// TIA Portal V15.1 export
// export: Created 2024-06-21T08:41:20.6972322Z, ExportSetting WithDefaults, DisplayName Totally Integrated Automation Portal, DisplayVersion V15.1 Update 5, DisplayName TIA Portal Openness, DisplayVersion V15.1 Update 5, DisplayName SINAMICS Startdrive Advanced, DisplayVersion V15.1, DisplayName G130, G150, S120, S150, SINAMICS MV, S210, DisplayVersion V15.1, DisplayName G110M, G120, G120C, G120D, G120P, DisplayVersion V15.1, DisplayName STEP 7 Professional, DisplayVersion V15.1 Update 5, DisplayName STEP 7 Safety, DisplayVersion V15.1, DisplayName WinCC Professional, DisplayVersion V15.1 Update 5, DisplayName SIMATIC Visualization Architect, DisplayVersion V15.1
FUNCTION_BLOCK "LCycleMonitoring"   // FB6056, FBD
TITLE = LCycleMonitoring - 2017/08/31
{ S7_Optimized_Access := 'FALSE' }
AUTHOR : hbracke
FAMILY : DataHand
VERSION : 0.1
// Used to monitor the cycle of a subzone and report the results to IT. On top it also creates an overtime alarm.
// stored: AutoNumber false, IsIECCheckEnabled false, SetENOAutomatically False, UDAEnableTagReadback false
   VAR_INPUT
      I_DateTimeFromPlc { ExternalAccessible := 'False'; ExternalVisible := 'False'; ExternalWritable := 'False'} : Date_And_Time;   // Actual Date and time from PLC
      I_PlcStatus { ExternalAccessible := 'False'; ExternalVisible := 'False'; ExternalWritable := 'False'} : DWord;   // Actual global PLC status
      I_ZmStatus { ExternalAccessible := 'False'; ExternalVisible := 'False'; ExternalWritable := 'False'} : "ZMStatus";   // Actual ModeZone status
      I_SubZoneStatus { ExternalAccessible := 'False'; ExternalVisible := 'False'; ExternalWritable := 'False'} : "SubzoneStatus";   // Actual status of one Subzone within the ModeZone
      I_OperatorStatus1 { ExternalAccessible := 'False'; ExternalVisible := 'False'; ExternalWritable := 'False'} : "OperatorStatus";   // Actual status of an operator
      I_OperatorStatus2 { ExternalAccessible := 'False'; ExternalVisible := 'False'; ExternalWritable := 'False'} : "OperatorStatus";   // Actual status of an operator
      I_OperatorStatus3 { ExternalAccessible := 'False'; ExternalVisible := 'False'; ExternalWritable := 'False'} : "OperatorStatus";   // Actual status of an operator
      I_OperatorStatus4 { ExternalAccessible := 'False'; ExternalVisible := 'False'; ExternalWritable := 'False'} : "OperatorStatus";   // Actual status of an operator
      I_OperatorStatus5 { ExternalAccessible := 'False'; ExternalVisible := 'False'; ExternalWritable := 'False'} : "OperatorStatus";   // Actual status of an operator
      I_OperatorStatus6 { ExternalAccessible := 'False'; ExternalVisible := 'False'; ExternalWritable := 'False'} : "OperatorStatus";   // Actual status of an operator
      I_PcsBodyId { ExternalAccessible := 'False'; ExternalVisible := 'False'; ExternalWritable := 'False'} : DWord;   // Body identification of in the SubZone; can be BodyNumber, Tagnumber, MixNumber or sequence number
      I_PcsBodyType { ExternalAccessible := 'False'; ExternalVisible := 'False'; ExternalWritable := 'False'} : DWord;   // Body type identification in Subzone
      I_RobotProgramNumber { ExternalAccessible := 'False'; ExternalVisible := 'False'; ExternalWritable := 'False'} : DWord;   // Program number of the robot
      I_CarrierId { ExternalAccessible := 'False'; ExternalVisible := 'False'; ExternalWritable := 'False'} : DWord;   // Identification of the carrier
      I_SubCarrierId { ExternalAccessible := 'False'; ExternalVisible := 'False'; ExternalWritable := 'False'} : DWord;   // Identification of a subcarrier
      I_AutoZoneReferenceCycle { ExternalAccessible := 'False'; ExternalVisible := 'False'; ExternalWritable := 'False'} : DWord;   // Reference cycle time for this zone for this product type
      I_Operator1RefCycle { ExternalAccessible := 'False'; ExternalVisible := 'False'; ExternalWritable := 'False'} : DWord;   // Reference cycle time for this zone for this product type
      I_Operator2RefCycle { ExternalAccessible := 'False'; ExternalVisible := 'False'; ExternalWritable := 'False'} : DWord;   // Reference cycle time for this zone for this product type
      I_Operator3RefCycle { ExternalAccessible := 'False'; ExternalVisible := 'False'; ExternalWritable := 'False'} : DWord;   // Reference cycle time for this zone for this product type
      I_Operator4RefCycle { ExternalAccessible := 'False'; ExternalVisible := 'False'; ExternalWritable := 'False'} : DWord;   // Reference cycle time for this zone for this product type
      I_Operator5RefCycle { ExternalAccessible := 'False'; ExternalVisible := 'False'; ExternalWritable := 'False'} : DWord;   // Reference cycle time for this zone for this product type
      I_Operator6RefCycle { ExternalAccessible := 'False'; ExternalVisible := 'False'; ExternalWritable := 'False'} : DWord;   // Reference cycle time for this zone for this product type
      C_StationNumber { ExternalAccessible := 'False'; ExternalVisible := 'False'; ExternalWritable := 'False'} : DWord;   // Station number (6 digits) where this subzone belongs to. Syntax is LLLSSS where LLL is the line number and SSS is the station number.
      C_ModeZoneNumber { ExternalAccessible := 'False'; ExternalVisible := 'False'; ExternalWritable := 'False'} : DWord;   // Number of the modezone. LLLSSSZMxx where xx is the number of the modezone.
      C_SubZoneNumber { ExternalAccessible := 'False'; ExternalVisible := 'False'; ExternalWritable := 'False'} : DWord;   // Is a number identifying the subzone within the Modezone. Syntax is mmx where mm is the number of the modezone and x is a sequencial number of the subzone.
      C_SubSystem { ExternalAccessible := 'False'; ExternalVisible := 'False'; ExternalWritable := 'False'} : Int;   // Number to identify the subsystem / Identify Subsystem / Identification of the Subsystem
      C_VDCommRecvDB { ExternalAccessible := 'False'; ExternalVisible := 'False'; ExternalWritable := 'False'} : DB_ANY;   // VD communication system receive DB; Not to be used by Application
      C_VDCommSendDB { ExternalAccessible := 'False'; ExternalVisible := 'False'; ExternalWritable := 'False'} : DB_ANY;   // VD communication system send DB; Not to be used by Application
      C_LocalRecvDB { ExternalAccessible := 'False'; ExternalVisible := 'False'; ExternalWritable := 'False'} : DB_ANY;   // Local DB For Recv Data Used By The Application
      C_LocalSendDB { ExternalAccessible := 'False'; ExternalVisible := 'False'; ExternalWritable := 'False'} : DB_ANY;   // Local DB For Send Data Used By The Application
   END_VAR
   VAR_OUTPUT
      O_WaitingInput { ExternalAccessible := 'False'; ExternalVisible := 'False'; ExternalWritable := 'False'} : Bool;   // Summary of waiting input status; any waiting input is active
      O_WaitingOutput { ExternalAccessible := 'False'; ExternalVisible := 'False'; ExternalWritable := 'False'} : Bool;   // Summary of waiting output status is active
      O_AutoZoneOverCycle { ExternalAccessible := 'False'; ExternalVisible := 'False'; ExternalWritable := 'False'} : Bool;   // Automatic unit has exceeded reference time
      O_Operator1OverCycle { ExternalAccessible := 'False'; ExternalVisible := 'False'; ExternalWritable := 'False'} : Bool;   // Operator has exceeded reference time
      O_Operator1OverCycleWarning { ExternalAccessible := 'False'; ExternalVisible := 'False'; ExternalWritable := 'False'} : Bool;   // Operator has exceeded 90% reference time
      O_Operator2OverCycle { ExternalAccessible := 'False'; ExternalVisible := 'False'; ExternalWritable := 'False'} : Bool;   // Operator has exceeded reference time
      O_Operator2OverCycleWarning { ExternalAccessible := 'False'; ExternalVisible := 'False'; ExternalWritable := 'False'} : Bool;   // Operator has exceeded 90% reference time
      O_Operator3OverCycle { ExternalAccessible := 'False'; ExternalVisible := 'False'; ExternalWritable := 'False'} : Bool;   // Operator has exceeded reference time
      O_Operator3OverCycleWarning { ExternalAccessible := 'False'; ExternalVisible := 'False'; ExternalWritable := 'False'} : Bool;   // Operator has exceeded 90% reference time
      O_Operator4OverCycle { ExternalAccessible := 'False'; ExternalVisible := 'False'; ExternalWritable := 'False'} : Bool;   // Operator has exceeded reference time
      O_Operator4OverCycleWarning { ExternalAccessible := 'False'; ExternalVisible := 'False'; ExternalWritable := 'False'} : Bool;   // Operator has exceeded 90% reference time
      O_Operator5OverCycle { ExternalAccessible := 'False'; ExternalVisible := 'False'; ExternalWritable := 'False'} : Bool;   // Operator has exceeded reference time
      O_Operator5OverCycleWarning { ExternalAccessible := 'False'; ExternalVisible := 'False'; ExternalWritable := 'False'} : Bool;   // Operator has exceeded 90% reference time
      O_Operator6OverCycle { ExternalAccessible := 'False'; ExternalVisible := 'False'; ExternalWritable := 'False'} : Bool;   // Operator has exceeded reference time
      O_Operator6OverCycleWarning { ExternalAccessible := 'False'; ExternalVisible := 'False'; ExternalWritable := 'False'} : Bool;   // Operator has exceeded 90% reference time
      O_WarningAlarm { ExternalAccessible := 'False'; ExternalVisible := 'False'; ExternalWritable := 'False'} : Bool;   // Summary of internal warning alarms
   END_VAR
   VAR_IN_OUT
      IO_VD : "VDComm";   // Signal handshake LVdComMaster
      IO_Modes : "Modes";   // Modes record to infeed the modes status of this subzone
      IO_Robot1 : "Robot";   // Robot record to exchange all robot statusses
      IO_Robot2 : "Robot";   // Robot record to exchange all robot statusses
      IO_Robot3 : "Robot";   // Robot record to exchange all robot statusses
      IO_Robot4 : "Robot";   // Robot record to exchange all robot statusses
      IO_Robot5 : "Robot";   // Robot record to exchange all robot statusses
      IO_Robot6 : "Robot";   // Robot record to exchange all robot statusses
      IO_Robot7 : "Robot";   // Robot record to exchange all robot statusses
      IO_Robot8 : "Robot";   // Robot record to exchange all robot statusses
      IO_Robot9 : "Robot";   // Robot record to exchange all robot statusses
      IO_Robot10 : "Robot";   // Robot record to exchange all robot statusses
      IO_Robot11 : "Robot";   // Robot record to exchange all robot statusses
      IO_Robot12 : "Robot";   // Robot record to exchange all robot statusses
      IO_Robot13 : "Robot";   // Robot record to exchange all robot statusses
      IO_Robot14 : "Robot";   // Robot record to exchange all robot statusses
      H_HMI : "H_HMI";   // HMI interface
      H_CycleMonitor : "H_CycleMonitoring";   // HMI interface
   END_VAR
   VAR DB_SPECIFIC
      DateTime { ExternalAccessible := 'False'; ExternalVisible := 'False'; ExternalWritable := 'False'} : Date_And_Time;   // Date and Time from the PLC. Each scan updated.
      SendToVD { ExternalAccessible := 'False'; ExternalVisible := 'False'; ExternalWritable := 'False'} : Bool;   // Trigger to send data to VD when Cycle is finished
      SendDoneVD { ExternalAccessible := 'False'; ExternalVisible := 'False'; ExternalWritable := 'False'} : Bool;   // Request Is Finished / Send operation is finished
      ResetVDComm { ExternalAccessible := 'False'; ExternalVisible := 'False'; ExternalWritable := 'False'} : Bool;   // Reset VD communication upon timeout
      InitState { ExternalAccessible := 'False'; ExternalVisible := 'False'; ExternalWritable := 'False'} : Bool;   // Flag indicating the initial run of the module
      StartOfCyclePulse { ExternalAccessible := 'False'; ExternalVisible := 'False'; ExternalWritable := 'False'} : Bool;   // Pulse at the start of a cycle
      EndOfCyclePulse { ExternalAccessible := 'False'; ExternalVisible := 'False'; ExternalWritable := 'False'} : Bool;   // Pulse at end of the cycle
      EndOfCycleReached { ExternalAccessible := 'False'; ExternalVisible := 'False'; ExternalWritable := 'False'} : Bool;   // Bit set to indicate the end of a cycle
      EndOfRecordReached { ExternalAccessible := 'False'; ExternalVisible := 'False'; ExternalWritable := 'False'} : Bool;   // Bit set when end of record was reached. A new record shall be setup
      AnyRobotActive { ExternalAccessible := 'False'; ExternalVisible := 'False'; ExternalWritable := 'False'} : Bool;   // Summary of all robots active
      AnyOperatorActive { ExternalAccessible := 'False'; ExternalVisible := 'False'; ExternalWritable := 'False'} : Bool;   // Summary of all operators active
      AnyOperatorOverCycle { ExternalAccessible := 'False'; ExternalVisible := 'False'; ExternalWritable := 'False'} : Bool;   // Summary of all operators
      StopActive { ExternalAccessible := 'False'; ExternalVisible := 'False'; ExternalWritable := 'False'} : Bool;   // Summery of all stopping conditions
      AutoZoneOverCycle { ExternalAccessible := 'False'; ExternalVisible := 'False'; ExternalWritable := 'False'} : Bool;   // Automatic zone is in over cycle
      WaitingInput { ExternalAccessible := 'False'; ExternalVisible := 'False'; ExternalWritable := 'False'} : Bool;   // Summary of all waiting input conditions
      WaitingOutput { ExternalAccessible := 'False'; ExternalVisible := 'False'; ExternalWritable := 'False'} : Bool;   // Summary of all waiting output conditions
      Operator1OverCycle { ExternalAccessible := 'False'; ExternalVisible := 'False'; ExternalWritable := 'False'} : Bool;   // Operator action exceeds reference tme
      Operator2OverCycle { ExternalAccessible := 'False'; ExternalVisible := 'False'; ExternalWritable := 'False'} : Bool;   // Operator action exceeds reference tme
      Operator3OverCycle { ExternalAccessible := 'False'; ExternalVisible := 'False'; ExternalWritable := 'False'} : Bool;   // Operator action exceeds reference tme
      Operator4OverCycle { ExternalAccessible := 'False'; ExternalVisible := 'False'; ExternalWritable := 'False'} : Bool;   // Operator action exceeds reference tme
      Operator5OverCycle { ExternalAccessible := 'False'; ExternalVisible := 'False'; ExternalWritable := 'False'} : Bool;   // Operator action exceeds reference tme
      Operator6OverCycle { ExternalAccessible := 'False'; ExternalVisible := 'False'; ExternalWritable := 'False'} : Bool;   // Operator action exceeds reference tme
      Operator1OverCycleWarning { ExternalAccessible := 'False'; ExternalVisible := 'False'; ExternalWritable := 'False'} : Bool;   // Operator action exceeds 90% of reference tme
      Operator2OverCycleWarning { ExternalAccessible := 'False'; ExternalVisible := 'False'; ExternalWritable := 'False'} : Bool;   // Operator action exceeds 90% of reference tme
      Operator3OverCycleWarning { ExternalAccessible := 'False'; ExternalVisible := 'False'; ExternalWritable := 'False'} : Bool;   // Operator action exceeds 90% of reference tme
      Operator4OverCycleWarning { ExternalAccessible := 'False'; ExternalVisible := 'False'; ExternalWritable := 'False'} : Bool;   // Operator action exceeds 90% of reference tme
      Operator5OverCycleWarning { ExternalAccessible := 'False'; ExternalVisible := 'False'; ExternalWritable := 'False'} : Bool;   // Operator action exceeds 90% of reference tme
      Operator6OverCycleWarning { ExternalAccessible := 'False'; ExternalVisible := 'False'; ExternalWritable := 'False'} : Bool;   // Operator action exceeds 90% of reference tme
      MaxRecordCountAlm { ExternalAccessible := 'False'; ExternalVisible := 'False'; ExternalWritable := 'False'} : Bool;   // Maximum amount of records within one cycle reported
      WarningAlarm { ExternalAccessible := 'False'; ExternalVisible := 'False'; ExternalWritable := 'False'} : Bool;   // Summary of warning alarms
      AlarmA { ExternalAccessible := 'False'; ExternalVisible := 'False'; ExternalWritable := 'False'} : Bool;   // Alarm A created by this function
      AlarmB { ExternalAccessible := 'False'; ExternalVisible := 'False'; ExternalWritable := 'False'} : Bool;   // Alarm B created by this function
      AlarmC { ExternalAccessible := 'False'; ExternalVisible := 'False'; ExternalWritable := 'False'} : Bool;   // Alarm C created by this function
      AlarmD { ExternalAccessible := 'False'; ExternalVisible := 'False'; ExternalWritable := 'False'} : Bool;   // Alarm D created by this function
      MaxIndex { ExternalAccessible := 'False'; ExternalVisible := 'False'; ExternalWritable := 'False'} : Int;   // Maximum value for Index
      Index { ExternalAccessible := 'False'; ExternalVisible := 'False'; ExternalWritable := 'False'} : Int;   // index to point to data values in event array
      MaxEofRecCounter { ExternalAccessible := 'False'; ExternalVisible := 'False'; ExternalWritable := 'False'} : Int;   // Maximum value that the record is allowed to loop without new start of cycle
      EofRecordCounter { ExternalAccessible := 'False'; ExternalVisible := 'False'; ExternalWritable := 'False'} : Int;   // Counting number of end of record events within 1 cycle
      SendLength { ExternalAccessible := 'False'; ExternalVisible := 'False'; ExternalWritable := 'False'} : Word;   // Pointer / Lenght of the data packet to be send
      VirtualBodyId { ExternalAccessible := 'False'; ExternalVisible := 'False'; ExternalWritable := 'False'} : DWord;   // Virtual created BodyId in case I_PcsBodyId is 0
      TotalProcessCycleTime { ExternalAccessible := 'False'; ExternalVisible := 'False'; ExternalWritable := 'False'} : Time;   // Accumulating timer (ms) to set the total cycle time
      TotalProcessWorkTime { ExternalAccessible := 'False'; ExternalVisible := 'False'; ExternalWritable := 'False'} : Time;   // Accumulating timer (ms) to set the total processwork time
      TotalOperator1Time { ExternalAccessible := 'False'; ExternalVisible := 'False'; ExternalWritable := 'False'} : Time;   // Accumulating timer (ms) of operator 1
      TotalOperator2Time { ExternalAccessible := 'False'; ExternalVisible := 'False'; ExternalWritable := 'False'} : Time;   // Accumulating timer (ms) of operator 2
      TotalOperator3Time { ExternalAccessible := 'False'; ExternalVisible := 'False'; ExternalWritable := 'False'} : Time;   // Accumulating timer (ms) of operator 3
      TotalOperator4Time { ExternalAccessible := 'False'; ExternalVisible := 'False'; ExternalWritable := 'False'} : Time;   // Accumulating timer (ms) of operator 4
      TotalOperator5Time { ExternalAccessible := 'False'; ExternalVisible := 'False'; ExternalWritable := 'False'} : Time;   // Accumulating timer (ms) of operator 5
      TotalOperator6Time { ExternalAccessible := 'False'; ExternalVisible := 'False'; ExternalWritable := 'False'} : Time;   // Accumulating timer (ms) of operator 6
      TotalWaitingInputTime { ExternalAccessible := 'False'; ExternalVisible := 'False'; ExternalWritable := 'False'} : Time;   // Accumulating timer (ms) to set the total waiting input time
      TotalInfeedTime { ExternalAccessible := 'False'; ExternalVisible := 'False'; ExternalWritable := 'False'} : Time;   // Accumulating timer (ms) to set the total Infeed time
      TotalWaitingOutputTime { ExternalAccessible := 'False'; ExternalVisible := 'False'; ExternalWritable := 'False'} : Time;   // Accumulating timer (ms) to set the total waiting output time
      TotalOutfeedTime { ExternalAccessible := 'False'; ExternalVisible := 'False'; ExternalWritable := 'False'} : Time;   // Accumulating timer (ms) to set the total Outfeed time
      TotalWaitingProcessWorkTime { ExternalAccessible := 'False'; ExternalVisible := 'False'; ExternalWritable := 'False'} : Time;   // Accumulating timer (ms) to set the total waiting process work time
      TotalWaitingRecoveryTime { ExternalAccessible := 'False'; ExternalVisible := 'False'; ExternalWritable := 'False'} : Time;   // Accumulating timer (ms) to set the total recovery time
      Memory { ExternalAccessible := 'False'; ExternalVisible := 'False'; ExternalWritable := 'False'} : Array[1..256] of Bool;   // Memory bits used to create edges
      CycleMonitorBuffer { ExternalAccessible := 'False'; ExternalVisible := 'False'; ExternalWritable := 'False'; S7_SetPoint := 'True'} : "H_CycleMonitoring";   // Array of display lines used as buffer
      CycleData { ExternalAccessible := 'False'; ExternalVisible := 'False'; ExternalWritable := 'False'; S7_SetPoint := 'True'} : "CycleTimeReportData";   // Record containing report Data
      CycleSendData { ExternalAccessible := 'False'; ExternalVisible := 'False'; ExternalWritable := 'False'; S7_SetPoint := 'True'} : "CycleTimeReportSendData";   // Record containing data to be send
   END_VAR
   VAR
      _LVDComSubSystem { ExternalAccessible := 'False'; ExternalVisible := 'False'; ExternalWritable := 'False'; S7_SetPoint := 'True'} : "LVDComSubSystemS7-1500";   // MultiInstance DB
   END_VAR
   VAR DB_SPECIFIC
      SendToVDTimeOut { ExternalAccessible := 'False'; ExternalVisible := 'False'; ExternalWritable := 'False'; S7_SetPoint := 'True'} : IEC_TIMER;   // Send to VD timeout
      CalculateTotalCycleTime { ExternalAccessible := 'False'; ExternalVisible := 'False'; ExternalWritable := 'False'; S7_SetPoint := 'True'} : TONR_TIME;   // Accumulation of cycle time
      CalculateTotalOperatorTime { ExternalAccessible := 'False'; ExternalVisible := 'False'; ExternalWritable := 'False'; S7_SetPoint := 'True'} : TONR_TIME;   // Accucmulution of operator time
      CalculateTotalWaitingInput { ExternalAccessible := 'False'; ExternalVisible := 'False'; ExternalWritable := 'False'; S7_SetPoint := 'True'} : TONR_TIME;   // Accumulation of waiting input
      CalculateTotalInfeedTime { ExternalAccessible := 'False'; ExternalVisible := 'False'; ExternalWritable := 'False'; S7_SetPoint := 'True'} : TONR_TIME;   // Accumulated infeed time
      CalculateTotalWaitingOutput { ExternalAccessible := 'False'; ExternalVisible := 'False'; ExternalWritable := 'False'; S7_SetPoint := 'True'} : TONR_TIME;   // Accumulation of waiting output
      CalculateTotalOutfeedTime { ExternalAccessible := 'False'; ExternalVisible := 'False'; ExternalWritable := 'False'; S7_SetPoint := 'True'} : TONR_TIME;   // Accumulated outfeed time
      CalcTotalProcessCycleTime { ExternalAccessible := 'False'; ExternalVisible := 'False'; ExternalWritable := 'False'; S7_SetPoint := 'True'} : IEC_TIMER;   // Function to calculate total ProductionCycle time
      CalcTotalProcessWorkTime { ExternalAccessible := 'False'; ExternalVisible := 'False'; ExternalWritable := 'False'; S7_SetPoint := 'True'} : IEC_TIMER;   // Function to calculate total ProcessWork time
      CalcTotalOperator1Time { ExternalAccessible := 'False'; ExternalVisible := 'False'; ExternalWritable := 'False'; S7_SetPoint := 'True'} : IEC_TIMER;   // function to calculate operator 1 time
      CalcTotalOperator2Time { ExternalAccessible := 'False'; ExternalVisible := 'False'; ExternalWritable := 'False'; S7_SetPoint := 'True'} : IEC_TIMER;   // function to calculate operator 2 time
      CalcTotalOperator3Time { ExternalAccessible := 'False'; ExternalVisible := 'False'; ExternalWritable := 'False'; S7_SetPoint := 'True'} : IEC_TIMER;   // function to calculate operator 3 time
      CalcTotalOperator4Time { ExternalAccessible := 'False'; ExternalVisible := 'False'; ExternalWritable := 'False'; S7_SetPoint := 'True'} : IEC_TIMER;   // function to calculate operator 4 time
      CalcTotalOperator5Time { ExternalAccessible := 'False'; ExternalVisible := 'False'; ExternalWritable := 'False'; S7_SetPoint := 'True'} : IEC_TIMER;   // function to calculate operator 5 time
      CalcTotalOperator6Time { ExternalAccessible := 'False'; ExternalVisible := 'False'; ExternalWritable := 'False'; S7_SetPoint := 'True'} : IEC_TIMER;   // function to calculate operator 6 time
      CalcTotalWaitingInput { ExternalAccessible := 'False'; ExternalVisible := 'False'; ExternalWritable := 'False'; S7_SetPoint := 'True'} : IEC_TIMER;
      CalcTotalWaitingOutput { ExternalAccessible := 'False'; ExternalVisible := 'False'; ExternalWritable := 'False'; S7_SetPoint := 'True'} : IEC_TIMER;
      CalcTotalWaitingProcessWorkTime { ExternalAccessible := 'False'; ExternalVisible := 'False'; ExternalWritable := 'False'; S7_SetPoint := 'True'} : IEC_TIMER;   // function to calculate the total waiting process time
      CalcTotalRecoveryTime { ExternalAccessible := 'False'; ExternalVisible := 'False'; ExternalWritable := 'False'; S7_SetPoint := 'True'} : IEC_TIMER;   // function to calculate the total waiting end of cycle time
   END_VAR
   VAR_TEMP
      Operator1RefCycleTemp : Real;   // Convert Operator Ref Cycle
      Operator1WarningRefTemp : Real;   // Calculation Warning Operator Ref Cycle
      Operator1WarningRef : DWord;   // Convert Warning Operator Ref Cycle
      Operator2RefCycleTemp : Real;   // Convert Operator Ref Cycle
      Operator2WarningRefTemp : Real;   // Calculation Warning Operator Ref Cycle
      Operator2WarningRef : DWord;   // Convert Warning Operator Ref Cycle
      Operator3RefCycleTemp : Real;   // Convert Operator Ref Cycle
      Operator3WarningRefTemp : Real;   // Calculation Warning Operator Ref Cycle
      Operator3WarningRef : DWord;   // Convert Warning Operator Ref Cycle
      Operator4RefCycleTemp : Real;   // Convert Operator Ref Cycle
      Operator4WarningRefTemp : Real;   // Calculation Warning Operator Ref Cycle
      Operator4WarningRef : DWord;   // Convert Warning Operator Ref Cycle
      Operator5RefCycleTemp : Real;   // Convert Operator Ref Cycle
      Operator5WarningRefTemp : Real;   // Calculation Warning Operator Ref Cycle
      Operator5WarningRef : DWord;   // Convert Warning Operator Ref Cycle
      Operator6RefCycleTemp : Real;   // Convert Operator Ref Cycle
      Operator6WarningRefTemp : Real;   // Calculation Warning Operator Ref Cycle
      Operator6WarningRef : DWord;   // Convert Warning Operator Ref Cycle
      PtrARECV : Any;   // Pointer to the Application receive DB
      RecvMessType : Int;   // Message type of the received data
      RecvSubSyst : Int;   // Subsystem target number
      RcvLength : Int;   // Length of received data
      RecvDBNbr : Int;   // Receive system DB Number
      SendDBNbr : Int;   // Send system DB Number
      LocalRecvDBNbr : Int;   // Receive DB Number Local by Application
      LocalSendDBNbr : Int;   // Send DB Number Local by Application
   END_VAR
   VAR_TEMP   // added for the SCL form of the ladder/FBD networks
      _w1 : Bool;
      _w2 : Bool;
      _w3 : Bool;
   END_VAR
BEGIN

NETWORK
TITLE = **** 1 - Inputs **** Load DB / **** 1 - Inputs **** Load DB number
// Load DB numbers to local variables from the Receive and Send DB from - VD Master - VD Subsystem
// Read DB Number Recv
      OPN   #C_VDCommRecvDB;
      L     DBNO;
      T     #RecvDBNbr;

// Read DB Number Send
      OPN   #C_VDCommSendDB;
      L     DBNO;
      T     #SendDBNbr;

// DB Number from VD Sub system
      OPN   #C_LocalRecvDB;
      L     DBNO;
      T     #LocalRecvDBNbr;

// Read DB Number Send
      OPN   #C_LocalSendDB;
      L     DBNO;
      T     #LocalSendDBNbr;

REGION Network 2: **** 1 - Inputs **** Set Max Values
   // MaxIndex is the maxmum index used to store the last event
   // [Index ] is used to mark end of record
   // MaxEofRecordCount is used to limit the maximum of records send within one production cycle.
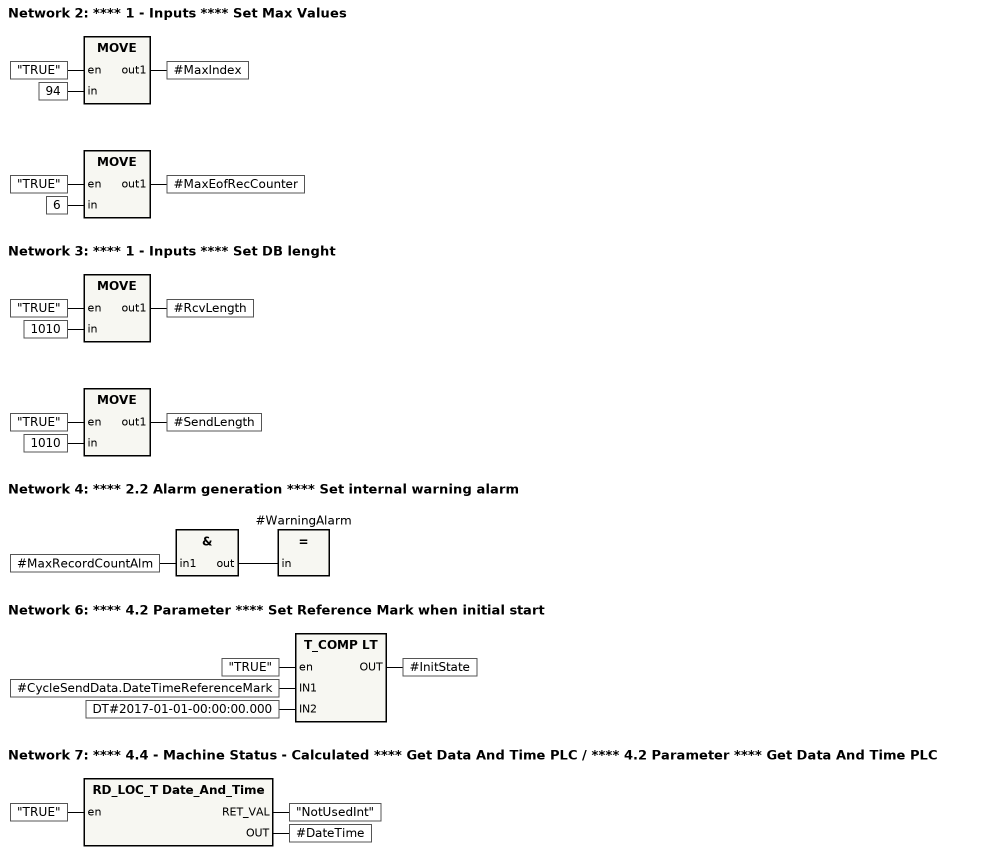
   IF "TRUE" THEN
       #MaxIndex := 94;
       #MaxEofRecCounter := 6;
   END_IF;
END_REGION

REGION Network 3: **** 1 - Inputs **** Set DB lenght
   // Set DB lenght. Make sure not to exceed the maximum TPDU size of one packet. 
   // Maximum size is 1024 - VD header (=10).
   // Lenght = Header (40) + ((MaxIndex + 2)*event lenght (10))
   IF "TRUE" THEN
       #RcvLength := 1010;
       #SendLength := 1010;
   END_IF;
END_REGION

REGION Network 4: **** 2.2 Alarm generation **** Set internal warning alarm
   #WarningAlarm := #MaxRecordCountAlm;
END_REGION

NETWORK
TITLE = **** 3.1 - Communication - Other Systems **** Configure DB / **** 4.2 Parameter **** Configure DB
// Configure DB pointers
      LAR1  P##PtrARECV;
      L     16#1002;  // Data type to copy B#16#2 = Bytes
      T     LW [AR1, P#0.0];
      L     #SendLength;  //Length sending data
      T     LW [AR1, P#2.0];
      L     #LocalSendDBNbr;  // Local Send DB Number
      T     LW [AR1, P#4.0];
      L     10;  // Offset in DB (skip VD header)
      SLD   3;  // Convert to pointer - Shift Left DW
      OD    16#8400_0000;  // Memory area DB Memory - 84 equals DB
      T     LD [AR1, P#6.0];


REGION Network 6: **** 4.2 Parameter **** Set Reference Mark when initial start
   // Check if reference mark has not been set, then initiate intial cycle.
   IF "TRUE" THEN
       T_COMP(IN1 := #CycleSendData.DateTimeReferenceMark, IN2 := DT#2017-01-01-00:00:00.000, OUT => #InitState);
   END_IF;
END_REGION

REGION Network 7: **** 4.4 - Machine Status - Calculated **** Get Data And Time PLC / **** 4.2 Parameter **** Get Data And Time PLC
   // Get Data And Time PLC / Get Data And Time PLC used to document the events.
   IF "TRUE" THEN "NotUsedInt" := RD_LOC_T(OUT => #DateTime); END_IF;
END_REGION

REGION Network 8: **** 3.1 - Communication - Other Systems **** MasterArea to SubArea / **** 4.4 Calculated **** MasterArea to SubArea - Set Reference Mark
   // Copy from MasterArea to SubArea
   // Copy Data from local stack to external VD DB
   // Set Bit to activate VD send procedure
   // Keep the SendToVd bit as long as procedure did not finish
   // Reset index pointer to start event storing in local stack
   // Reset trigger flags
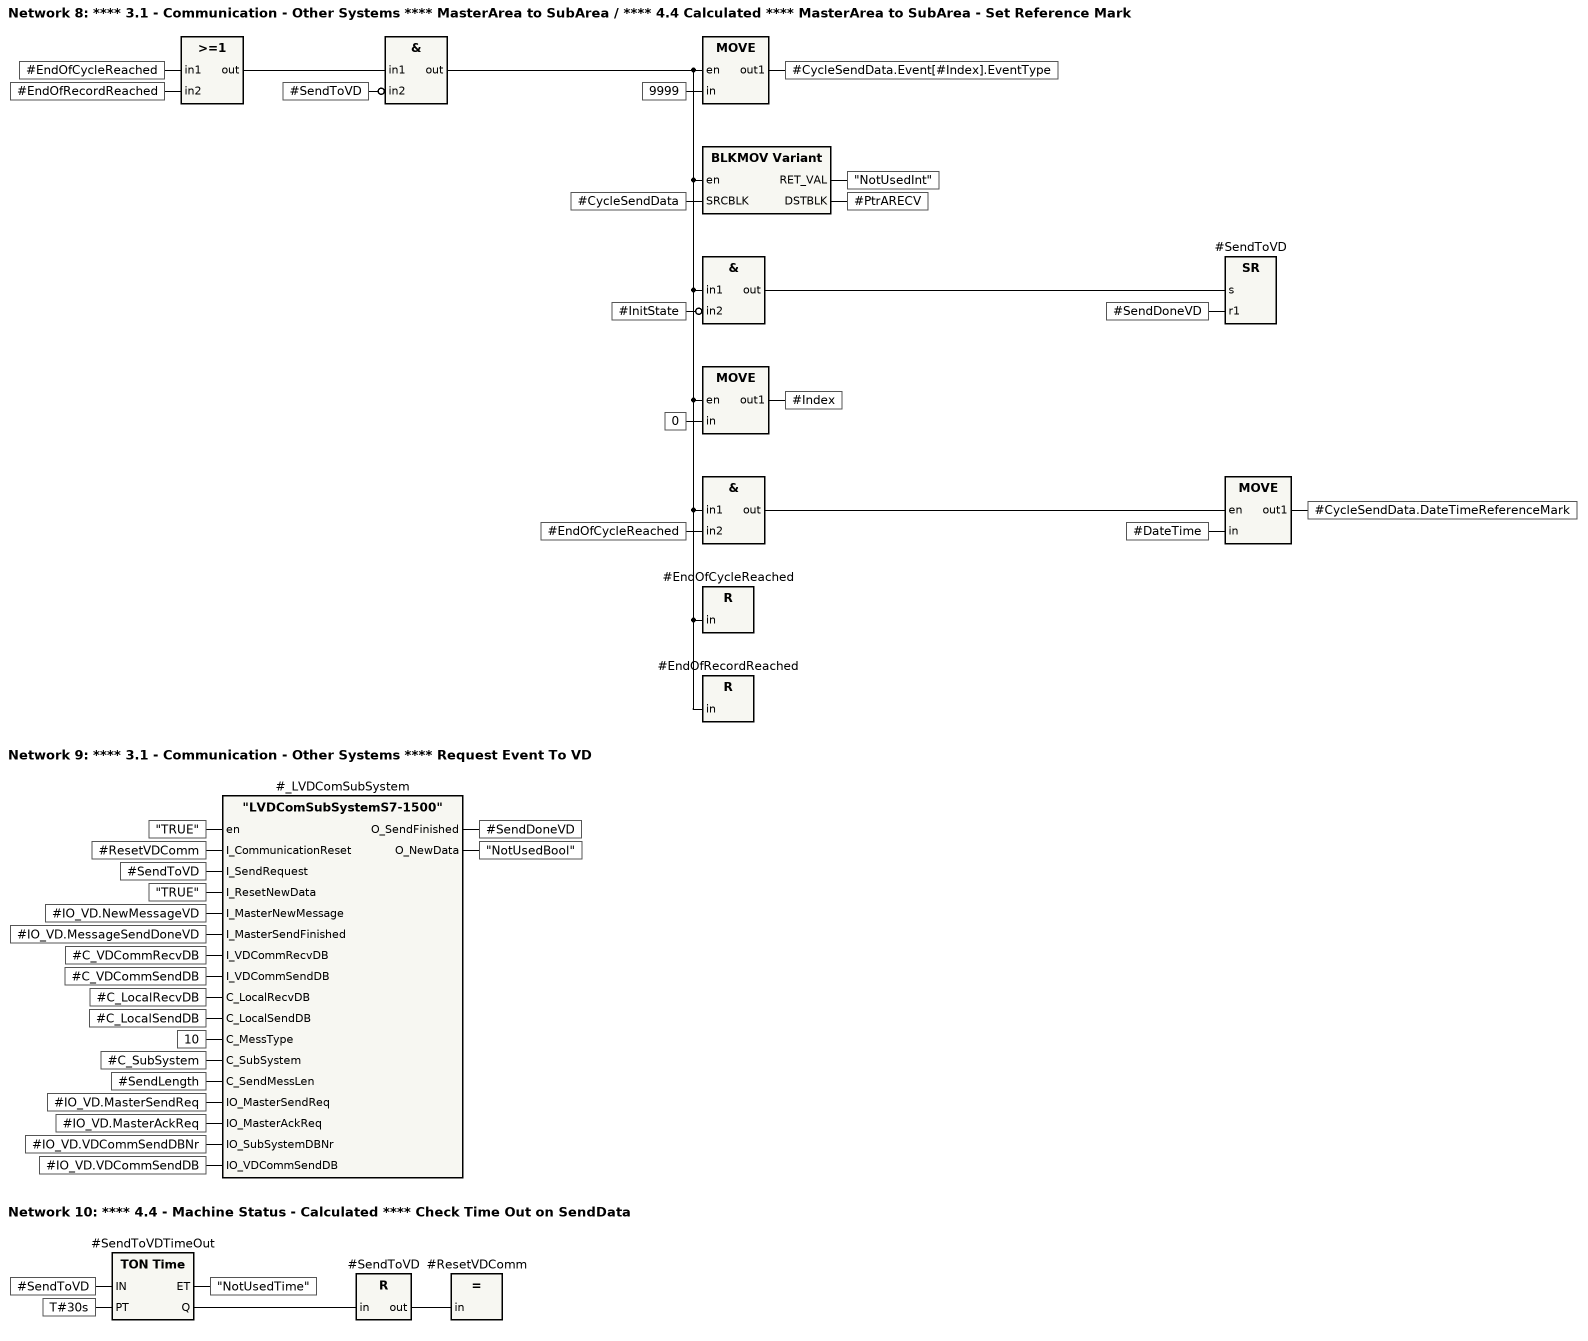
   #_w1 := (#EndOfCycleReached OR #EndOfRecordReached) AND NOT #SendToVD;
   IF #_w1 THEN
       #CycleSendData.Event[#Index].EventType := 9999;
       "NotUsedInt" := BLKMOV(SRCBLK := #CycleSendData, DSTBLK => #PtrARECV);
   END_IF;
   IF #_w1 AND NOT #InitState THEN
       #SendToVD := TRUE;   // SR flip-flop
   END_IF;
   IF #SendDoneVD THEN #SendToVD := FALSE; END_IF;
   IF #_w1 THEN #Index := 0; END_IF;
   IF #_w1 AND #EndOfCycleReached THEN #CycleSendData.DateTimeReferenceMark := #DateTime; END_IF;
   IF #_w1 THEN
       #EndOfCycleReached := FALSE;
       #EndOfRecordReached := FALSE;
   END_IF;
END_REGION

REGION Network 9: **** 3.1 - Communication - Other Systems **** Request Event To VD
   // Request Send To VD
   IF "TRUE" THEN
       #_LVDComSubSystem(I_CommunicationReset := #ResetVDComm,   // "LVDComSubSystemS7-1500"
                         I_SendRequest := #SendToVD,
                         I_ResetNewData := "TRUE",
                         I_MasterNewMessage := #IO_VD.NewMessageVD,
                         I_MasterSendFinished := #IO_VD.MessageSendDoneVD,
                         I_VDCommRecvDB := #C_VDCommRecvDB,
                         I_VDCommSendDB := #C_VDCommSendDB,
                         C_LocalRecvDB := #C_LocalRecvDB,
                         C_LocalSendDB := #C_LocalSendDB,
                         C_MessType := 10,
                         C_SubSystem := #C_SubSystem,
                         C_SendMessLen := #SendLength,
                         IO_MasterSendReq := #IO_VD.MasterSendReq,
                         IO_MasterAckReq := #IO_VD.MasterAckReq,
                         IO_SubSystemDBNr := #IO_VD.VDCommSendDBNr,
                         IO_VDCommSendDB := #IO_VD.VDCommSendDB,
                         O_SendFinished => #SendDoneVD,
                         O_NewData => "NotUsedBool");
   END_IF;
END_REGION

REGION Network 10: **** 4.4 - Machine Status - Calculated **** Check Time Out on SendData
   // Reset Send request when time out elapses
   // Reset the VD communication
   #SendToVDTimeOut.TON(IN := #SendToVD, PT := T#30s, ET => "NotUsedTime");
   IF #SendToVDTimeOut.Q THEN #SendToVD := FALSE; END_IF;
   #ResetVDComm := #SendToVDTimeOut.Q;
END_REGION

REGION Network 11: **** 4.4 - Machine Status - Calculated **** If maximum index is reached
   // Reset index when index is higher then MaxIndex or below zero.
   // Prevent illegal values
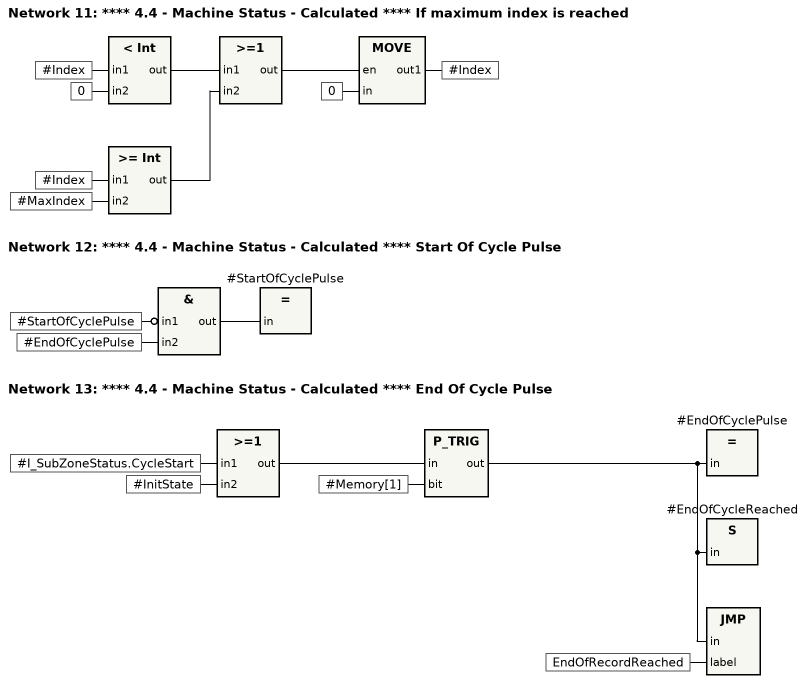
   IF (#Index < 0) OR (#Index >= #MaxIndex) THEN #Index := 0; END_IF;
END_REGION

REGION Network 12: **** 4.4 - Machine Status - Calculated **** Start Of Cycle Pulse
   // This is the trigger for the start of the production cycle
   // Trigger is created subsequent to the end of cycle
   #StartOfCyclePulse := NOT #StartOfCyclePulse AND #EndOfCyclePulse;
END_REGION

REGION Network 13: **** 4.4 - Machine Status - Calculated **** End Of Cycle Pulse
   // This is the trigger for the end of the production cycle
   #_w1 := #I_SubZoneStatus.CycleStart OR #InitState;
   #_w2 := #_w1 AND NOT #Memory[1];   // rising edge
   #Memory[1] := #_w1;
   #EndOfCyclePulse := #_w2;
   IF #_w2 THEN
       #EndOfCycleReached := TRUE;
       GOTO EndOfRecordReached;
   END_IF;
END_REGION

REGION Network 14: **** 4.4 - Machine Status - Calculated **** At the start of cycle
   // At the start of the production cycle, data of this cycle is initialised
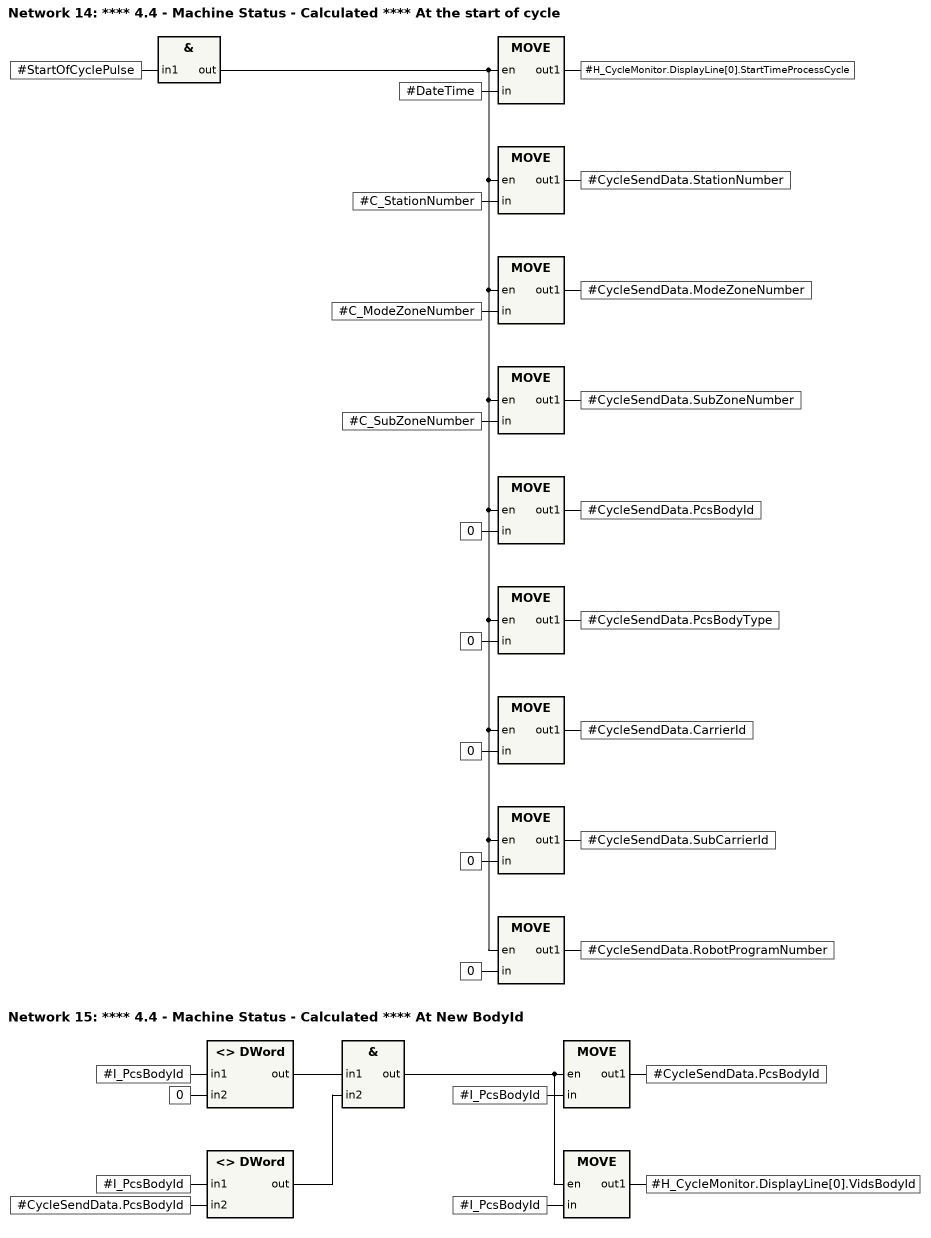
   IF #StartOfCyclePulse THEN
       #H_CycleMonitor.DisplayLine[0].StartTimeProcessCycle := #DateTime;
       #CycleSendData.StationNumber := #C_StationNumber;
       #CycleSendData.ModeZoneNumber := #C_ModeZoneNumber;
       #CycleSendData.SubZoneNumber := #C_SubZoneNumber;
       #CycleSendData.PcsBodyId := 0;
       #CycleSendData.PcsBodyType := 0;
       #CycleSendData.CarrierId := 0;
       #CycleSendData.SubCarrierId := 0;
       #CycleSendData.RobotProgramNumber := 0;
   END_IF;
END_REGION

REGION Network 15: **** 4.4 - Machine Status - Calculated **** At New BodyId
   // Copy BodyId at the moment the data is updated and different from 0
   #_w1 := (#I_PcsBodyId <> 0) AND (#I_PcsBodyId <> #CycleSendData.PcsBodyId);
   IF #_w1 THEN
       #CycleSendData.PcsBodyId := #I_PcsBodyId;
       #H_CycleMonitor.DisplayLine[0].VidsBodyId := #I_PcsBodyId;
   END_IF;
END_REGION

REGION Network 16: **** 4.4 - Machine Status - Calculated **** At New BodyType
   // Copy BodyType at the moment the data is updated and different from 0
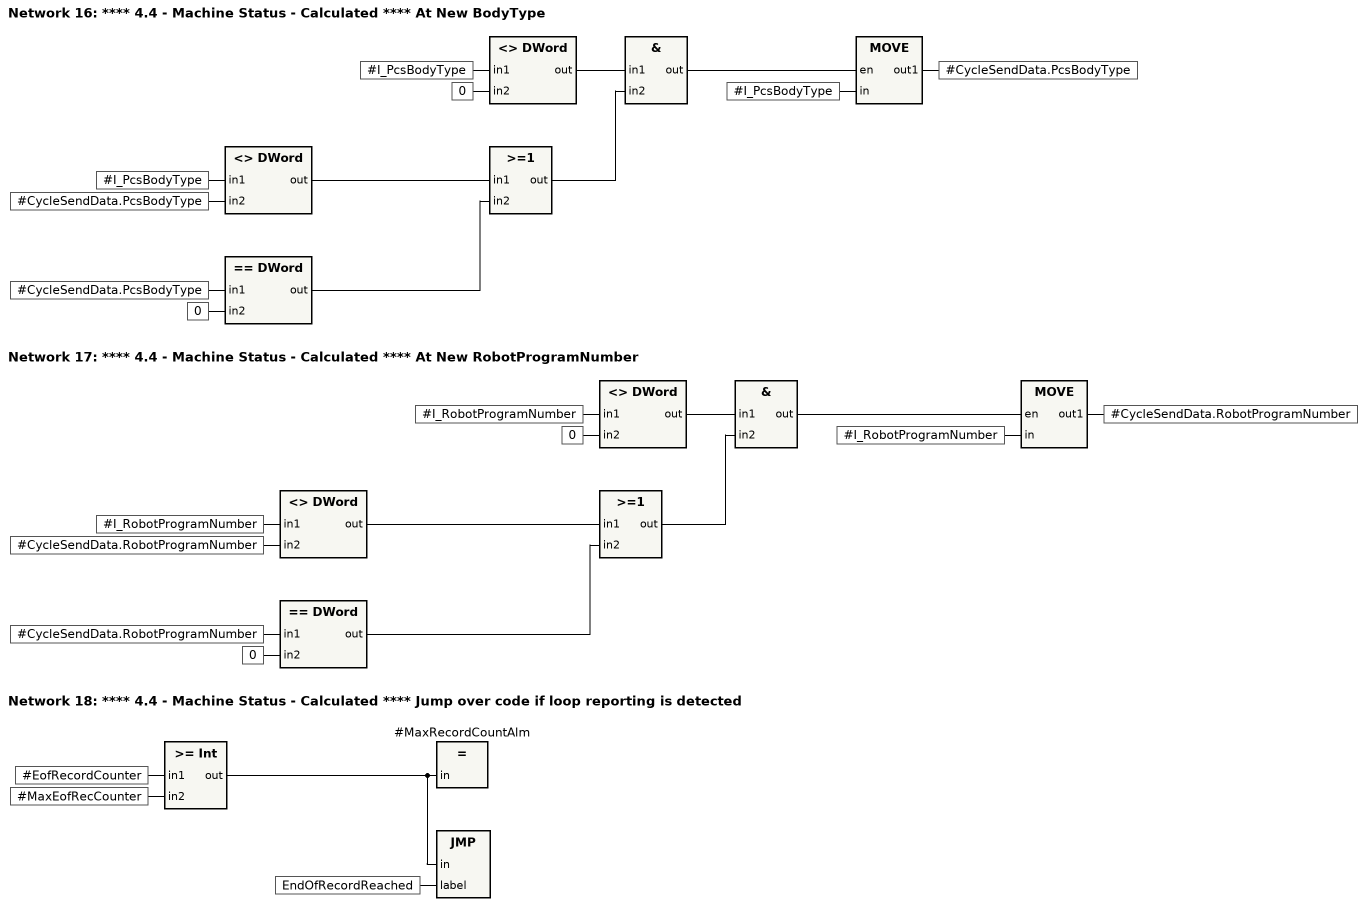
   IF (#I_PcsBodyType <> 0) AND ((#I_PcsBodyType <> #CycleSendData.PcsBodyType) OR (#CycleSendData.PcsBodyType = 0)) THEN
       #CycleSendData.PcsBodyType := #I_PcsBodyType;
   END_IF;
END_REGION

REGION Network 17: **** 4.4 - Machine Status - Calculated **** At New RobotProgramNumber
   // Copy BodyRobotProgramNumber at the moment the data is updated and different from 0
   IF (#I_RobotProgramNumber <> 0) AND ((#I_RobotProgramNumber <> #CycleSendData.RobotProgramNumber) OR (#CycleSendData.RobotProgramNumber = 0)) THEN
       #CycleSendData.RobotProgramNumber := #I_RobotProgramNumber;
   END_IF;
END_REGION

REGION Network 18: **** 4.4 - Machine Status - Calculated **** Jump over code if loop reporting is detected
   // When too many records are send within one production cycle then the reporting is ceesed. This to prevent that endless loops are overflowing the reporting database.
   // Reporting will resume at the next Start of Outfeed action.
   #MaxRecordCountAlm := #EofRecordCounter >= #MaxEofRecCounter;
   IF #MaxRecordCountAlm THEN GOTO EndOfRecordReached; END_IF;
END_REGION

REGION Network 19: **** 4.4 - Machine Status - Calculated **** Register Time events - BreakActive Start/stop
   // Create event
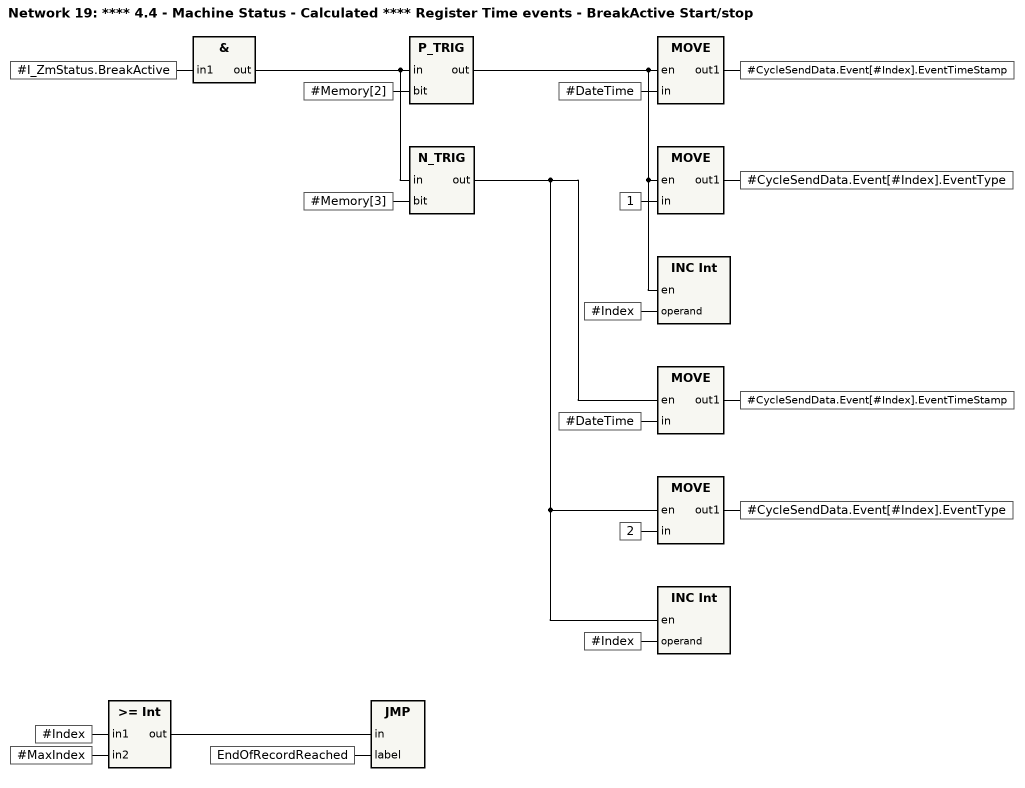
   #_w1 := #I_ZmStatus.BreakActive AND NOT #Memory[2];   // rising edge
   #Memory[2] := #I_ZmStatus.BreakActive;
   IF #_w1 THEN
       #CycleSendData.Event[#Index].EventTimeStamp := #DateTime;
       #CycleSendData.Event[#Index].EventType := 1;
       #Index := #Index + 1;
   END_IF;
   #_w2 := NOT #I_ZmStatus.BreakActive AND #Memory[3];   // falling edge
   #Memory[3] := #I_ZmStatus.BreakActive;
   IF #_w2 THEN
       #CycleSendData.Event[#Index].EventTimeStamp := #DateTime;
       #CycleSendData.Event[#Index].EventType := 2;
       #Index := #Index + 1;
   END_IF;
   IF #Index >= #MaxIndex THEN GOTO EndOfRecordReached; END_IF;
END_REGION

REGION Network 20: **** 4.4 - Machine Status - Calculated **** Register Time events - ProductionStop Start/stop
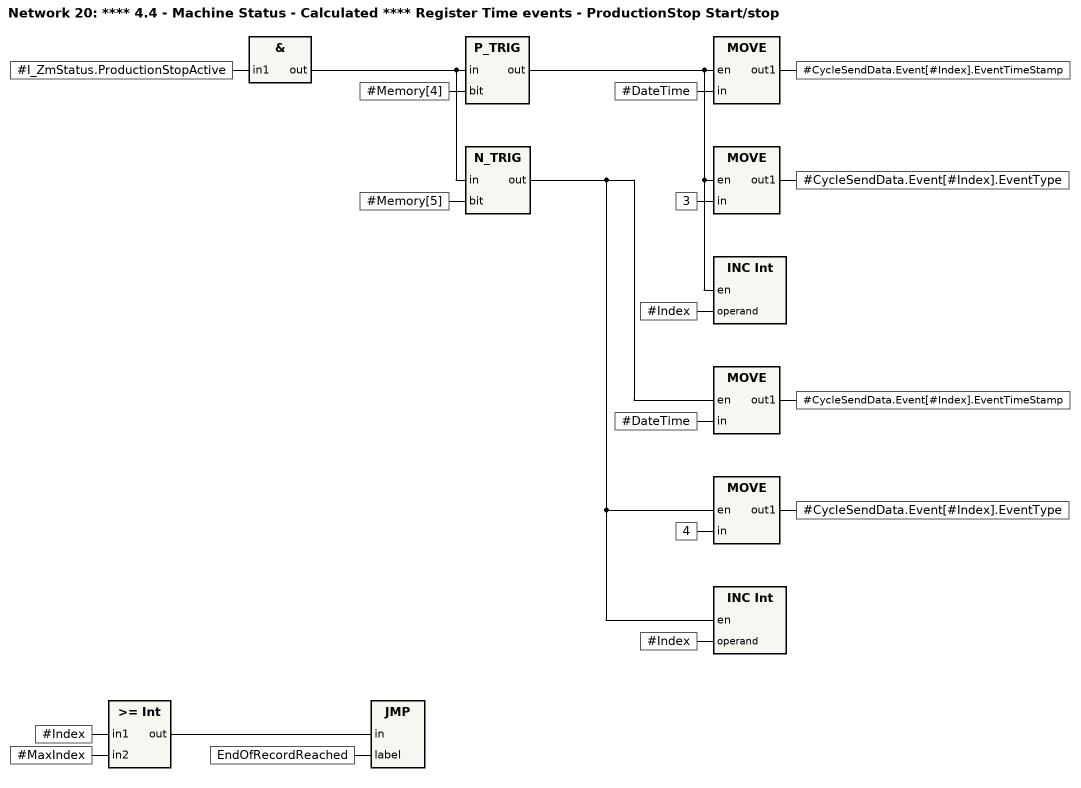
   #_w1 := #I_ZmStatus.ProductionStopActive AND NOT #Memory[4];   // rising edge
   #Memory[4] := #I_ZmStatus.ProductionStopActive;
   IF #_w1 THEN
       #CycleSendData.Event[#Index].EventTimeStamp := #DateTime;
       #CycleSendData.Event[#Index].EventType := 3;
       #Index := #Index + 1;
   END_IF;
   #_w2 := NOT #I_ZmStatus.ProductionStopActive AND #Memory[5];   // falling edge
   #Memory[5] := #I_ZmStatus.ProductionStopActive;
   IF #_w2 THEN
       #CycleSendData.Event[#Index].EventTimeStamp := #DateTime;
       #CycleSendData.Event[#Index].EventType := 4;
       #Index := #Index + 1;
   END_IF;
   IF #Index >= #MaxIndex THEN GOTO EndOfRecordReached; END_IF;
END_REGION

REGION Network 21: **** 4.4 - Machine Status - Calculated **** Register Time events - Service Start/stop
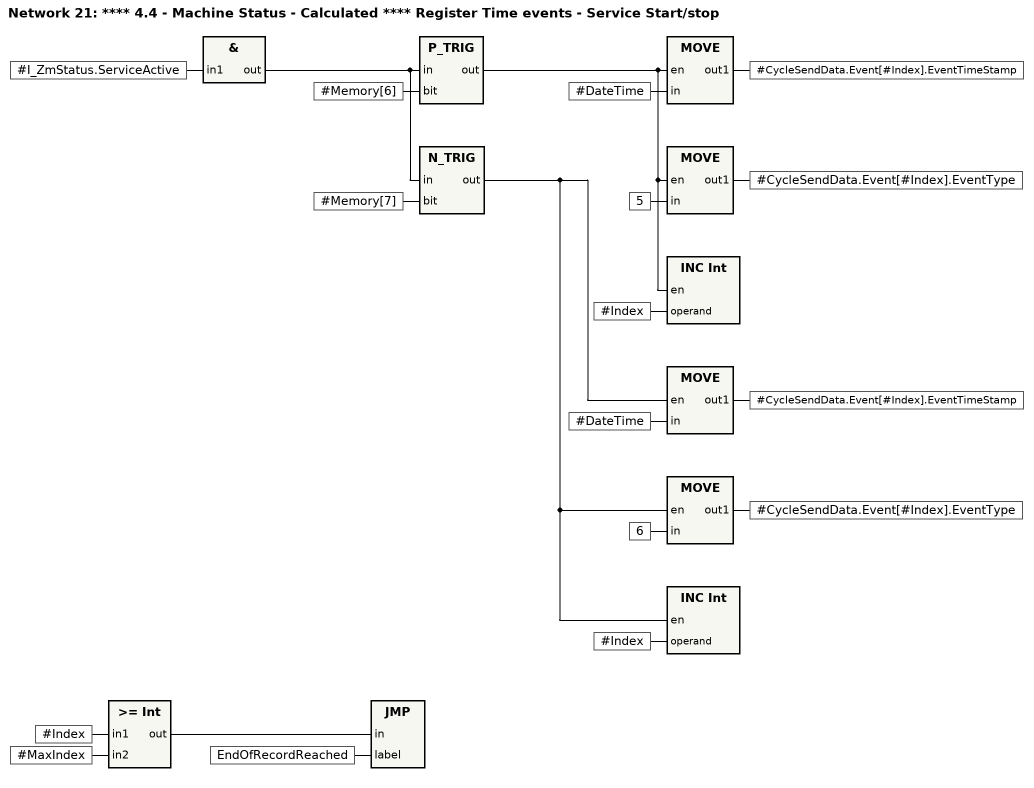
   #_w1 := #I_ZmStatus.ServiceActive AND NOT #Memory[6];   // rising edge
   #Memory[6] := #I_ZmStatus.ServiceActive;
   IF #_w1 THEN
       #CycleSendData.Event[#Index].EventTimeStamp := #DateTime;
       #CycleSendData.Event[#Index].EventType := 5;
       #Index := #Index + 1;
   END_IF;
   #_w2 := NOT #I_ZmStatus.ServiceActive AND #Memory[7];   // falling edge
   #Memory[7] := #I_ZmStatus.ServiceActive;
   IF #_w2 THEN
       #CycleSendData.Event[#Index].EventTimeStamp := #DateTime;
       #CycleSendData.Event[#Index].EventType := 6;
       #Index := #Index + 1;
   END_IF;
   IF #Index >= #MaxIndex THEN GOTO EndOfRecordReached; END_IF;
END_REGION

REGION Network 22: **** 4.4 - Machine Status - Calculated **** Register Time events - Maintenance Start/stop
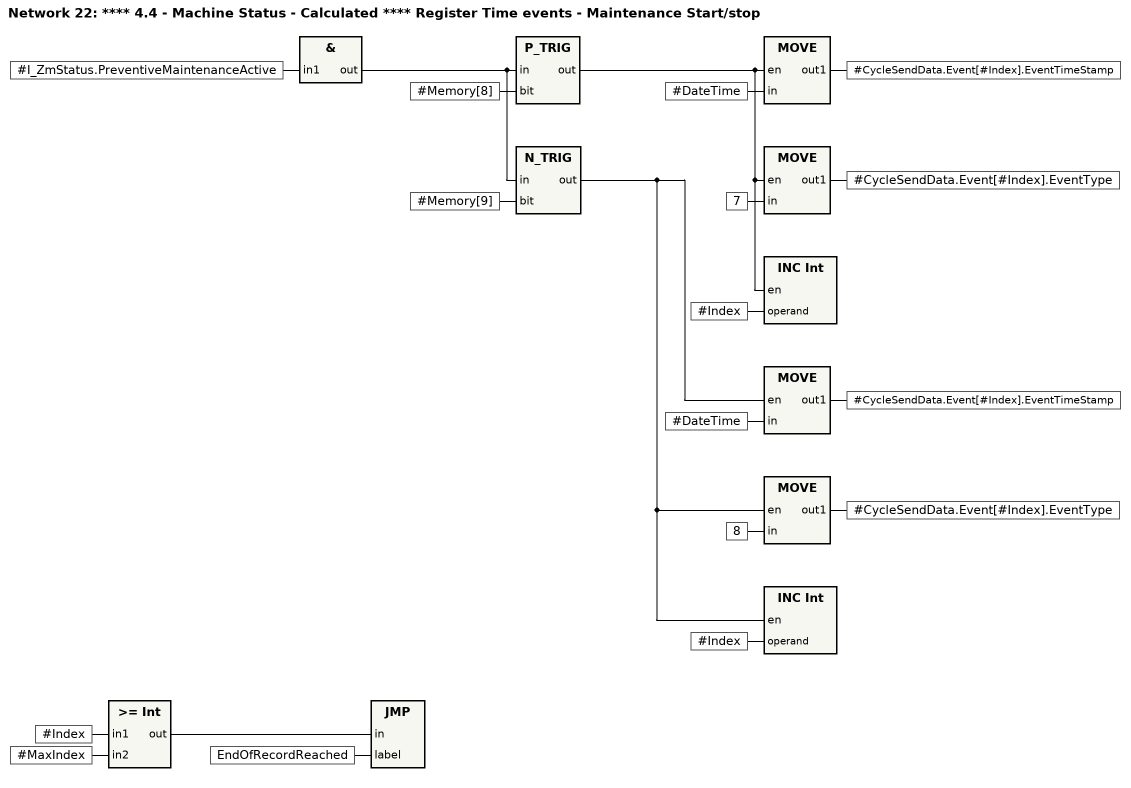
   #_w1 := #I_ZmStatus.PreventiveMaintenanceActive AND NOT #Memory[8];   // rising edge
   #Memory[8] := #I_ZmStatus.PreventiveMaintenanceActive;
   IF #_w1 THEN
       #CycleSendData.Event[#Index].EventTimeStamp := #DateTime;
       #CycleSendData.Event[#Index].EventType := 7;
       #Index := #Index + 1;
   END_IF;
   #_w2 := NOT #I_ZmStatus.PreventiveMaintenanceActive AND #Memory[9];   // falling edge
   #Memory[9] := #I_ZmStatus.PreventiveMaintenanceActive;
   IF #_w2 THEN
       #CycleSendData.Event[#Index].EventTimeStamp := #DateTime;
       #CycleSendData.Event[#Index].EventType := 8;
       #Index := #Index + 1;
   END_IF;
   IF #Index >= #MaxIndex THEN GOTO EndOfRecordReached; END_IF;
END_REGION

REGION Network 23: **** 4.4 - Machine Status - Calculated **** Register Time events - TeamMeeting Start/stop
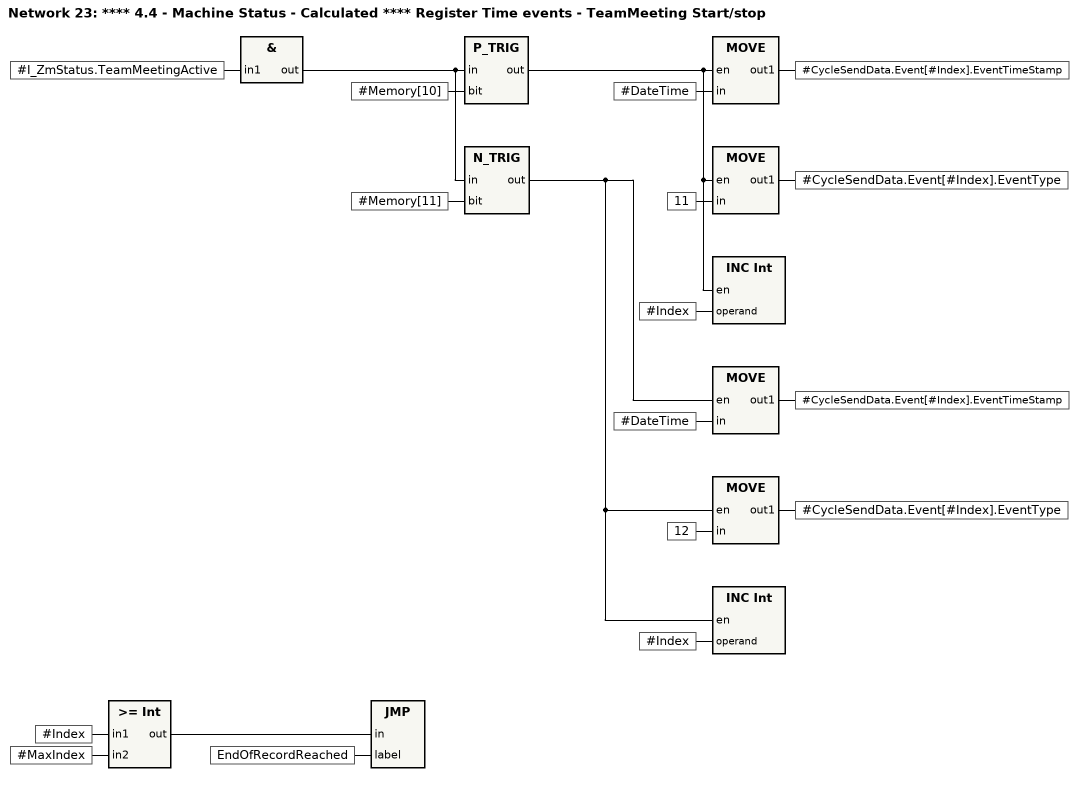
   #_w1 := #I_ZmStatus.TeamMeetingActive AND NOT #Memory[10];   // rising edge
   #Memory[10] := #I_ZmStatus.TeamMeetingActive;
   IF #_w1 THEN
       #CycleSendData.Event[#Index].EventTimeStamp := #DateTime;
       #CycleSendData.Event[#Index].EventType := 11;
       #Index := #Index + 1;
   END_IF;
   #_w2 := NOT #I_ZmStatus.TeamMeetingActive AND #Memory[11];   // falling edge
   #Memory[11] := #I_ZmStatus.TeamMeetingActive;
   IF #_w2 THEN
       #CycleSendData.Event[#Index].EventTimeStamp := #DateTime;
       #CycleSendData.Event[#Index].EventType := 12;
       #Index := #Index + 1;
   END_IF;
   IF #Index >= #MaxIndex THEN GOTO EndOfRecordReached; END_IF;
END_REGION

REGION Network 24: **** 4.4 - Machine Status - Calculated **** Register Time events - StoppingAlarmZm Start/stop
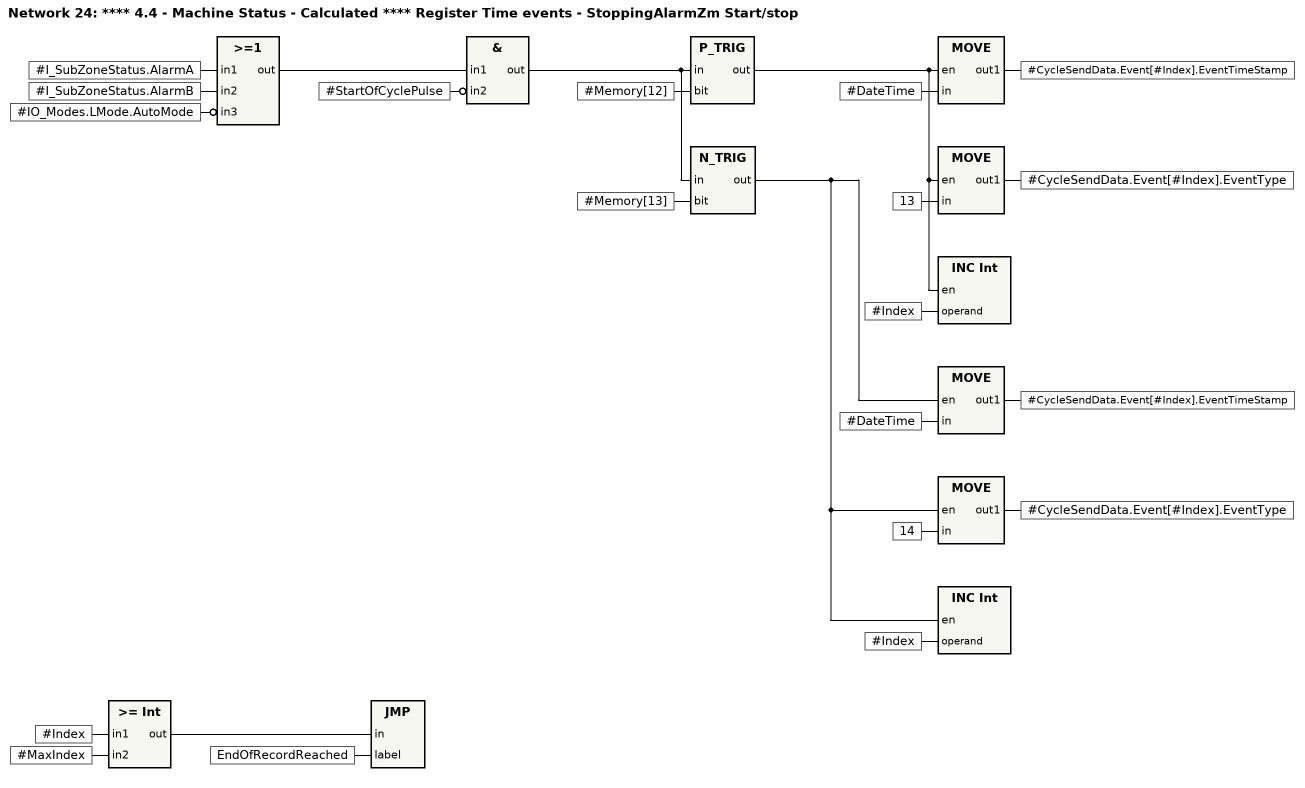
   #_w1 := (#I_SubZoneStatus.AlarmA OR #I_SubZoneStatus.AlarmB OR NOT #IO_Modes.LMode.AutoMode) AND NOT #StartOfCyclePulse;
   #_w2 := #_w1 AND NOT #Memory[12];   // rising edge
   #Memory[12] := #_w1;
   IF #_w2 THEN
       #CycleSendData.Event[#Index].EventTimeStamp := #DateTime;
       #CycleSendData.Event[#Index].EventType := 13;
       #Index := #Index + 1;
   END_IF;
   #_w3 := NOT #_w1 AND #Memory[13];   // falling edge
   #Memory[13] := #_w1;
   IF #_w3 THEN
       #CycleSendData.Event[#Index].EventTimeStamp := #DateTime;
       #CycleSendData.Event[#Index].EventType := 14;
       #Index := #Index + 1;
   END_IF;
   IF #Index >= #MaxIndex THEN GOTO EndOfRecordReached; END_IF;
END_REGION

REGION Network 25: **** 4.4 - Machine Status - Calculated **** Register Time events - WarningAlarmZm Start/stop
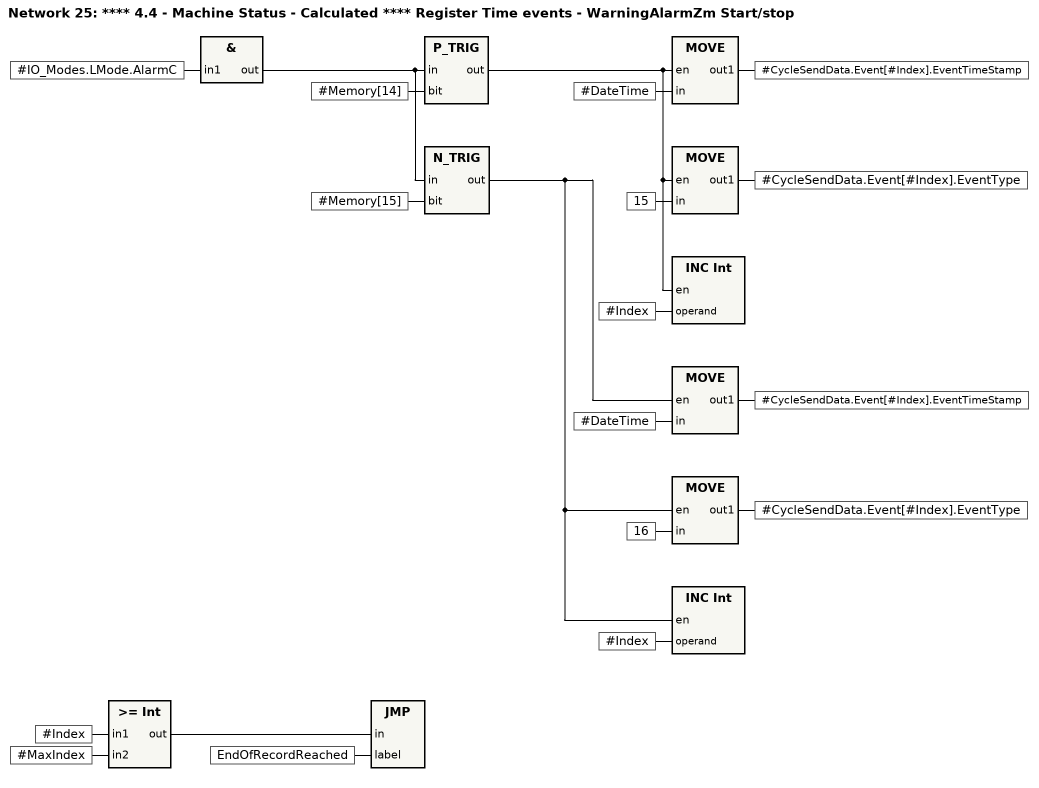
   #_w1 := #IO_Modes.LMode.AlarmC AND NOT #Memory[14];   // rising edge
   #Memory[14] := #IO_Modes.LMode.AlarmC;
   IF #_w1 THEN
       #CycleSendData.Event[#Index].EventTimeStamp := #DateTime;
       #CycleSendData.Event[#Index].EventType := 15;
       #Index := #Index + 1;
   END_IF;
   #_w2 := NOT #IO_Modes.LMode.AlarmC AND #Memory[15];   // falling edge
   #Memory[15] := #IO_Modes.LMode.AlarmC;
   IF #_w2 THEN
       #CycleSendData.Event[#Index].EventTimeStamp := #DateTime;
       #CycleSendData.Event[#Index].EventType := 16;
       #Index := #Index + 1;
   END_IF;
   IF #Index >= #MaxIndex THEN GOTO EndOfRecordReached; END_IF;
END_REGION

REGION Network 26: **** 4.4 - Machine Status - Calculated **** Register Time events - StoppingAlarmZms Start/stop
   // Alarm reported as long as AlarmABC is TRUE.
   // Resend alarm report at start of every cycle.
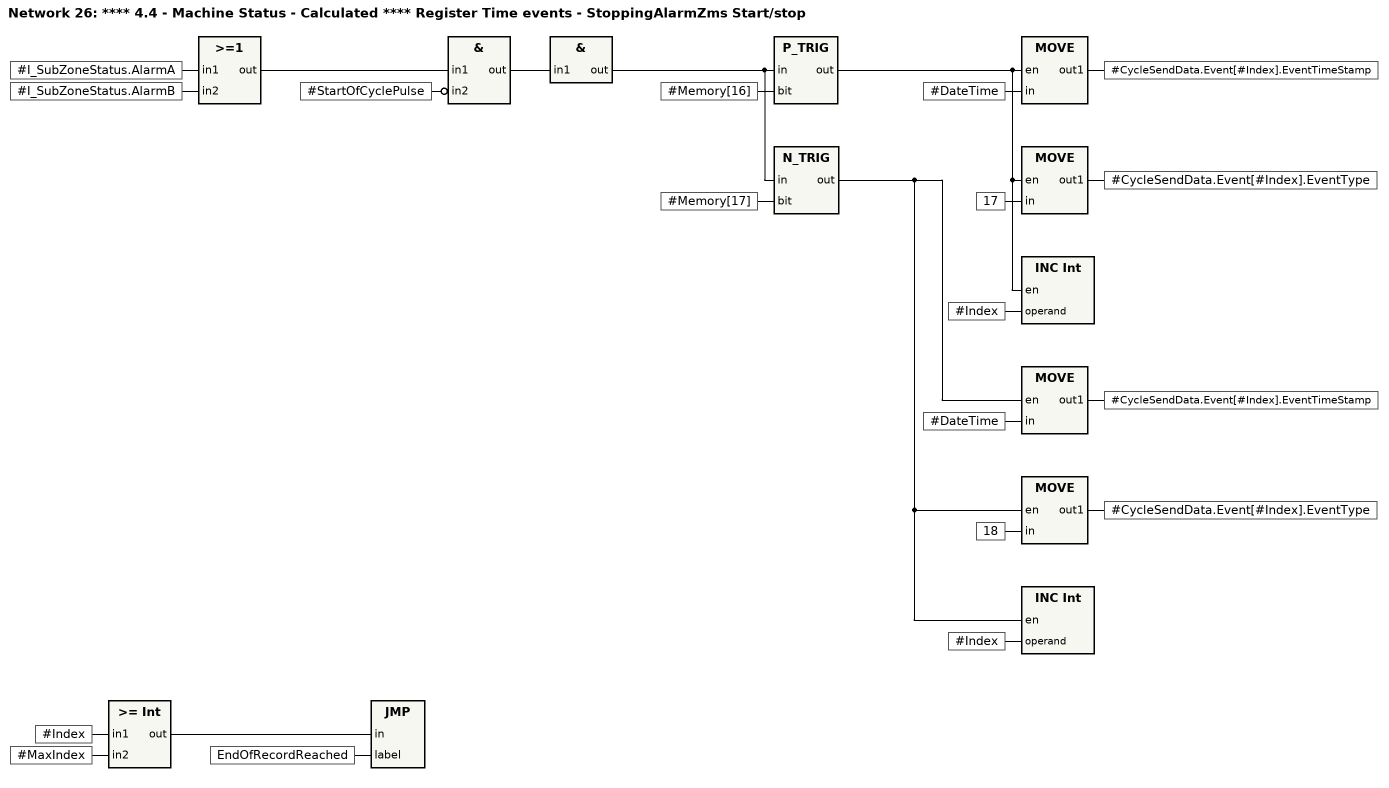
   #_w1 := (#I_SubZoneStatus.AlarmA OR #I_SubZoneStatus.AlarmB) AND NOT #StartOfCyclePulse;
   #_w2 := #_w1 AND NOT #Memory[16];   // rising edge
   #Memory[16] := #_w1;
   IF #_w2 THEN
       #CycleSendData.Event[#Index].EventTimeStamp := #DateTime;
       #CycleSendData.Event[#Index].EventType := 17;
       #Index := #Index + 1;
   END_IF;
   #_w3 := NOT #_w1 AND #Memory[17];   // falling edge
   #Memory[17] := #_w1;
   IF #_w3 THEN
       #CycleSendData.Event[#Index].EventTimeStamp := #DateTime;
       #CycleSendData.Event[#Index].EventType := 18;
       #Index := #Index + 1;
   END_IF;
   IF #Index >= #MaxIndex THEN GOTO EndOfRecordReached; END_IF;
END_REGION

REGION Network 27: **** 4.4 - Machine Status - Calculated **** Register Time events - WarningAlarmZms Start/stop
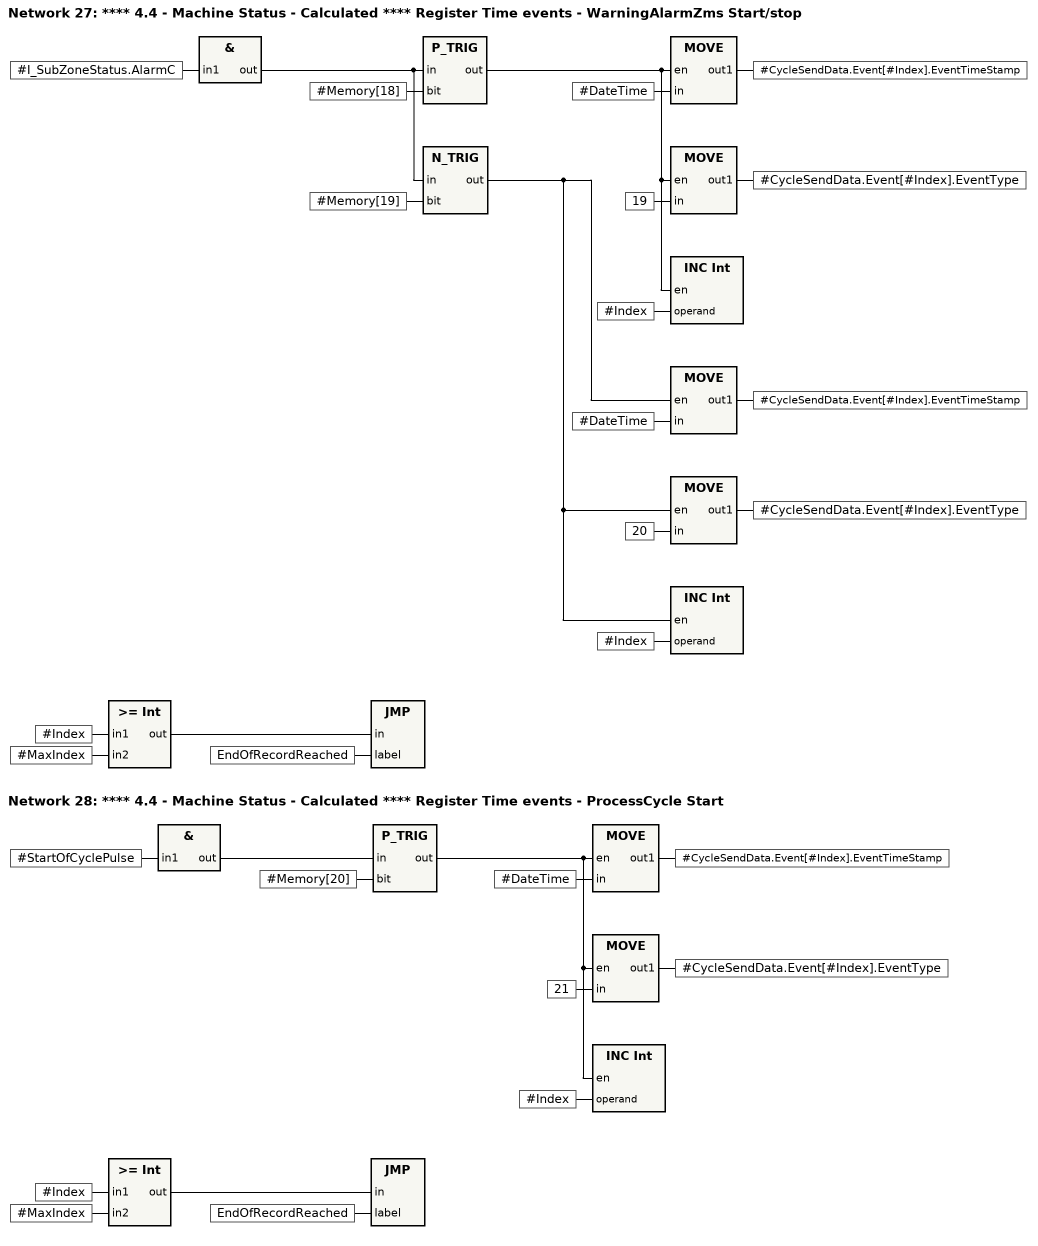
   #_w1 := #I_SubZoneStatus.AlarmC AND NOT #Memory[18];   // rising edge
   #Memory[18] := #I_SubZoneStatus.AlarmC;
   IF #_w1 THEN
       #CycleSendData.Event[#Index].EventTimeStamp := #DateTime;
       #CycleSendData.Event[#Index].EventType := 19;
       #Index := #Index + 1;
   END_IF;
   #_w2 := NOT #I_SubZoneStatus.AlarmC AND #Memory[19];   // falling edge
   #Memory[19] := #I_SubZoneStatus.AlarmC;
   IF #_w2 THEN
       #CycleSendData.Event[#Index].EventTimeStamp := #DateTime;
       #CycleSendData.Event[#Index].EventType := 20;
       #Index := #Index + 1;
   END_IF;
   IF #Index >= #MaxIndex THEN GOTO EndOfRecordReached; END_IF;
END_REGION

REGION Network 28: **** 4.4 - Machine Status - Calculated **** Register Time events - ProcessCycle Start
   #_w1 := #StartOfCyclePulse AND NOT #Memory[20];   // rising edge
   #Memory[20] := #StartOfCyclePulse;
   IF #_w1 THEN
       #CycleSendData.Event[#Index].EventTimeStamp := #DateTime;
       #CycleSendData.Event[#Index].EventType := 21;
       #Index := #Index + 1;
   END_IF;
   IF #Index >= #MaxIndex THEN GOTO EndOfRecordReached; END_IF;
END_REGION

REGION Network 29: **** 4.4 - Machine Status - Calculated **** Register Time events - WaitingInput1 Start/stop
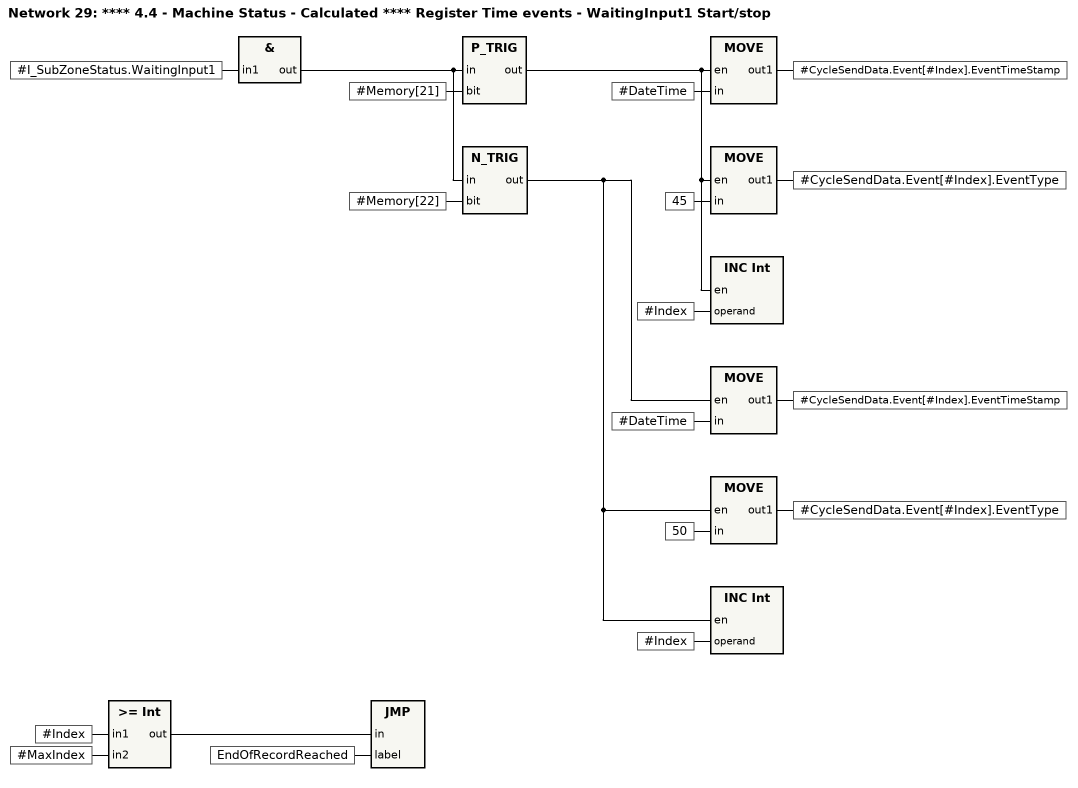
   #_w1 := #I_SubZoneStatus.WaitingInput1 AND NOT #Memory[21];   // rising edge
   #Memory[21] := #I_SubZoneStatus.WaitingInput1;
   IF #_w1 THEN
       #CycleSendData.Event[#Index].EventTimeStamp := #DateTime;
       #CycleSendData.Event[#Index].EventType := 45;
       #Index := #Index + 1;
   END_IF;
   #_w2 := NOT #I_SubZoneStatus.WaitingInput1 AND #Memory[22];   // falling edge
   #Memory[22] := #I_SubZoneStatus.WaitingInput1;
   IF #_w2 THEN
       #CycleSendData.Event[#Index].EventTimeStamp := #DateTime;
       #CycleSendData.Event[#Index].EventType := 50;
       #Index := #Index + 1;
   END_IF;
   IF #Index >= #MaxIndex THEN GOTO EndOfRecordReached; END_IF;
END_REGION

REGION Network 30: **** 4.4 - Machine Status - Calculated **** Register Time events - WaitingInput2 Start/stop
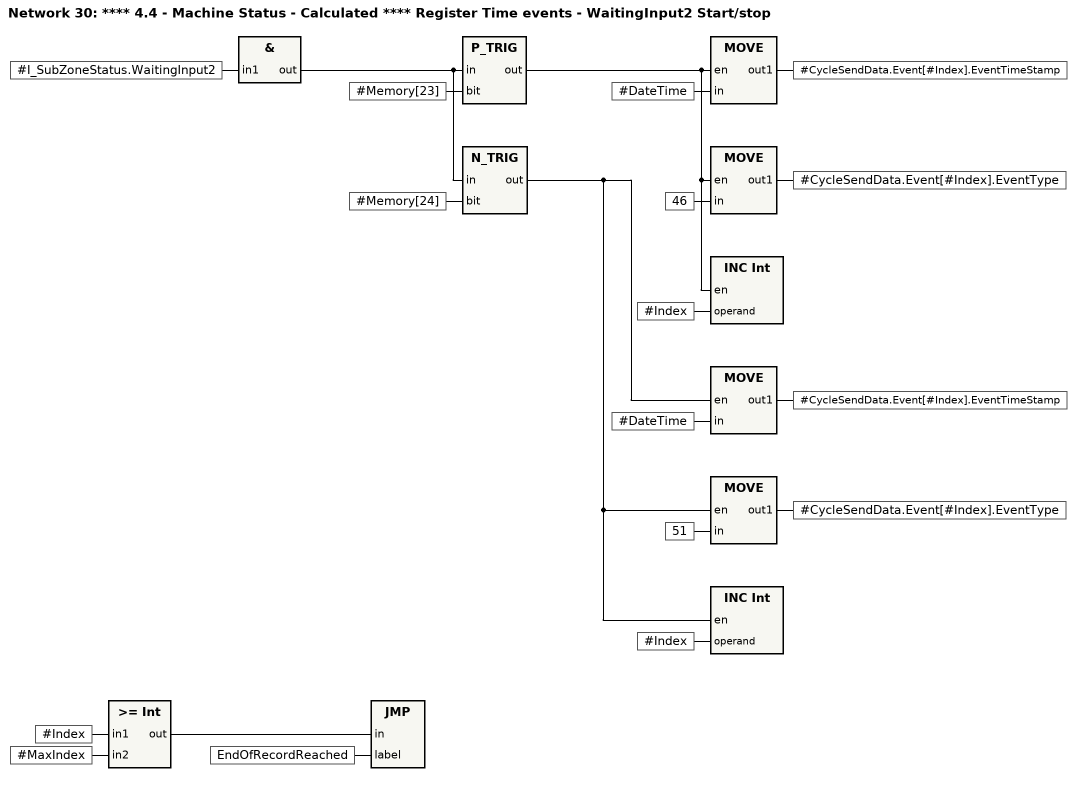
   #_w1 := #I_SubZoneStatus.WaitingInput2 AND NOT #Memory[23];   // rising edge
   #Memory[23] := #I_SubZoneStatus.WaitingInput2;
   IF #_w1 THEN
       #CycleSendData.Event[#Index].EventTimeStamp := #DateTime;
       #CycleSendData.Event[#Index].EventType := 46;
       #Index := #Index + 1;
   END_IF;
   #_w2 := NOT #I_SubZoneStatus.WaitingInput2 AND #Memory[24];   // falling edge
   #Memory[24] := #I_SubZoneStatus.WaitingInput2;
   IF #_w2 THEN
       #CycleSendData.Event[#Index].EventTimeStamp := #DateTime;
       #CycleSendData.Event[#Index].EventType := 51;
       #Index := #Index + 1;
   END_IF;
   IF #Index >= #MaxIndex THEN GOTO EndOfRecordReached; END_IF;
END_REGION

REGION Network 31: **** 4.4 - Machine Status - Calculated **** Register Time events - WaitingInput3 Start/stop
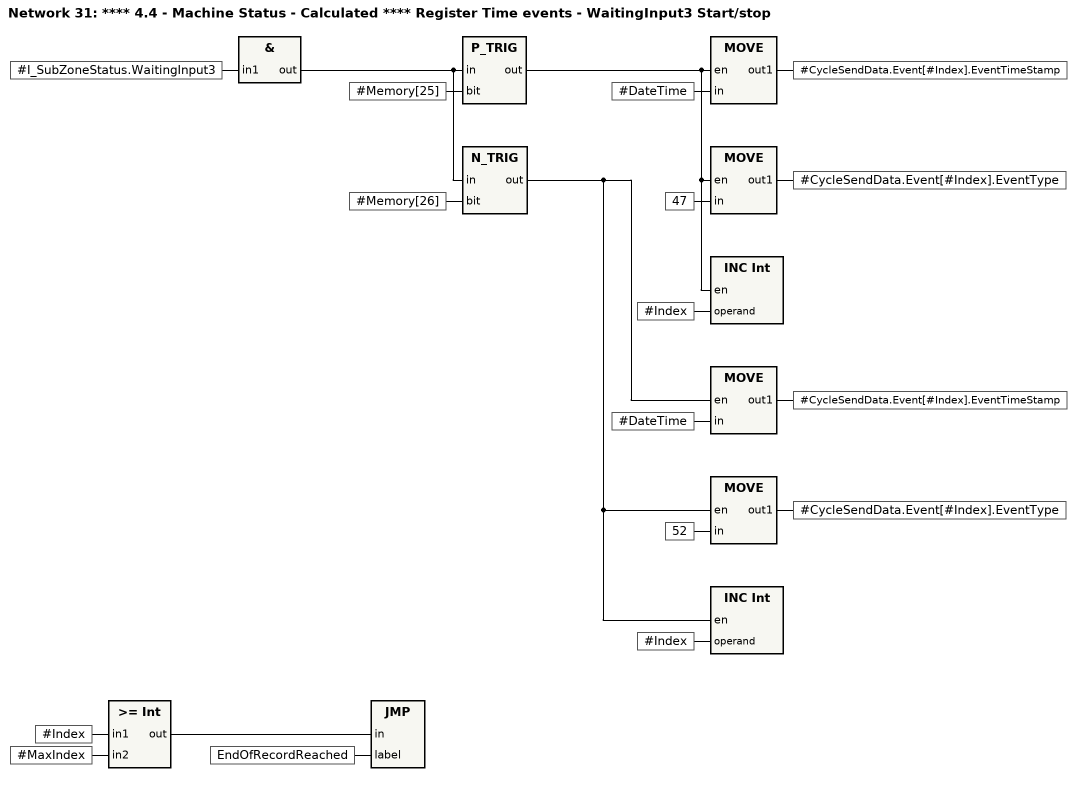
   #_w1 := #I_SubZoneStatus.WaitingInput3 AND NOT #Memory[25];   // rising edge
   #Memory[25] := #I_SubZoneStatus.WaitingInput3;
   IF #_w1 THEN
       #CycleSendData.Event[#Index].EventTimeStamp := #DateTime;
       #CycleSendData.Event[#Index].EventType := 47;
       #Index := #Index + 1;
   END_IF;
   #_w2 := NOT #I_SubZoneStatus.WaitingInput3 AND #Memory[26];   // falling edge
   #Memory[26] := #I_SubZoneStatus.WaitingInput3;
   IF #_w2 THEN
       #CycleSendData.Event[#Index].EventTimeStamp := #DateTime;
       #CycleSendData.Event[#Index].EventType := 52;
       #Index := #Index + 1;
   END_IF;
   IF #Index >= #MaxIndex THEN GOTO EndOfRecordReached; END_IF;
END_REGION

REGION Network 32: **** 4.4 - Machine Status - Calculated **** Register Time events - WaitingInput4 Start/stop
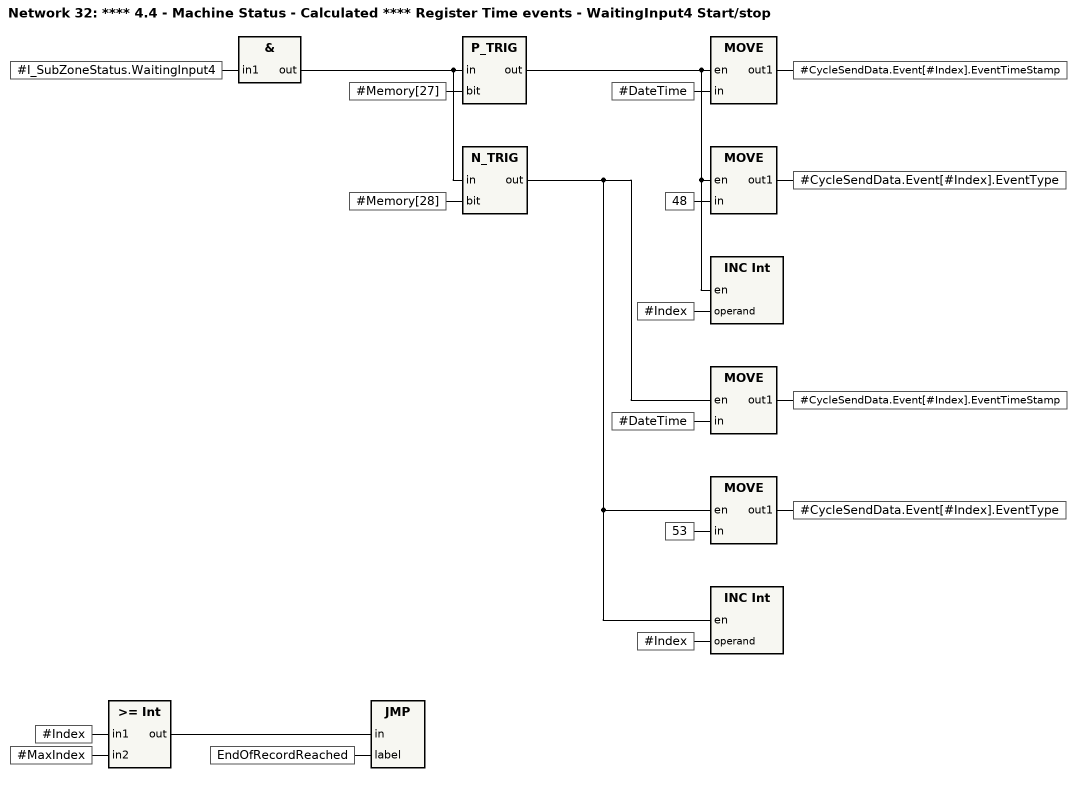
   #_w1 := #I_SubZoneStatus.WaitingInput4 AND NOT #Memory[27];   // rising edge
   #Memory[27] := #I_SubZoneStatus.WaitingInput4;
   IF #_w1 THEN
       #CycleSendData.Event[#Index].EventTimeStamp := #DateTime;
       #CycleSendData.Event[#Index].EventType := 48;
       #Index := #Index + 1;
   END_IF;
   #_w2 := NOT #I_SubZoneStatus.WaitingInput4 AND #Memory[28];   // falling edge
   #Memory[28] := #I_SubZoneStatus.WaitingInput4;
   IF #_w2 THEN
       #CycleSendData.Event[#Index].EventTimeStamp := #DateTime;
       #CycleSendData.Event[#Index].EventType := 53;
       #Index := #Index + 1;
   END_IF;
   IF #Index >= #MaxIndex THEN GOTO EndOfRecordReached; END_IF;
END_REGION

REGION Network 33: **** 4.4 - Machine Status - Calculated **** Register Time events - WaitingInput5 Start/stop
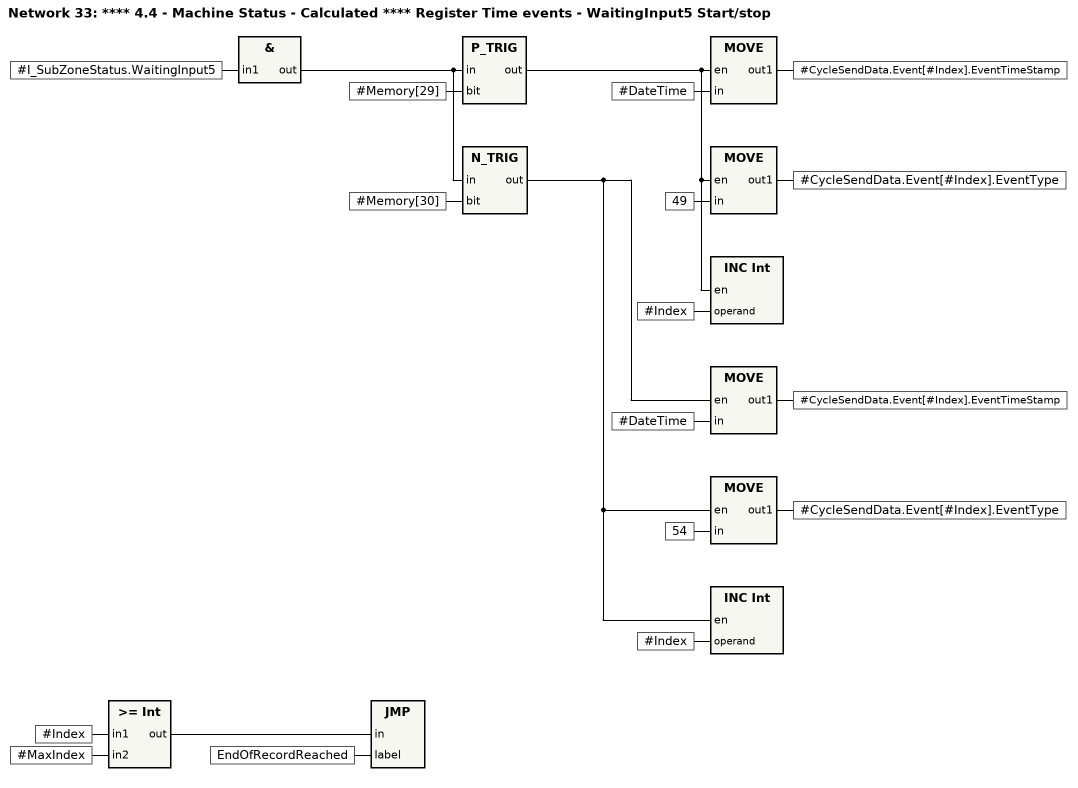
   #_w1 := #I_SubZoneStatus.WaitingInput5 AND NOT #Memory[29];   // rising edge
   #Memory[29] := #I_SubZoneStatus.WaitingInput5;
   IF #_w1 THEN
       #CycleSendData.Event[#Index].EventTimeStamp := #DateTime;
       #CycleSendData.Event[#Index].EventType := 49;
       #Index := #Index + 1;
   END_IF;
   #_w2 := NOT #I_SubZoneStatus.WaitingInput5 AND #Memory[30];   // falling edge
   #Memory[30] := #I_SubZoneStatus.WaitingInput5;
   IF #_w2 THEN
       #CycleSendData.Event[#Index].EventTimeStamp := #DateTime;
       #CycleSendData.Event[#Index].EventType := 54;
       #Index := #Index + 1;
   END_IF;
   IF #Index >= #MaxIndex THEN GOTO EndOfRecordReached; END_IF;
END_REGION

REGION Network 34: **** 4.4 - Machine Status - Calculated **** Register Time events - Infeed1 Start/stop
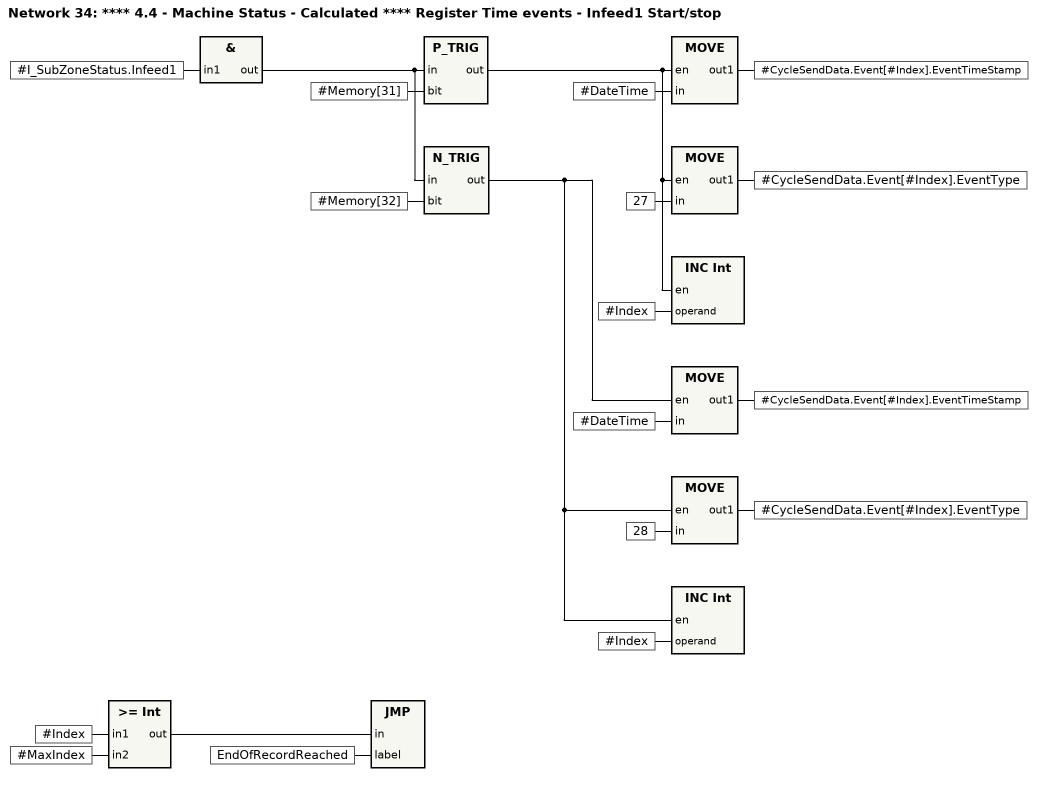
   #_w1 := #I_SubZoneStatus.Infeed1 AND NOT #Memory[31];   // rising edge
   #Memory[31] := #I_SubZoneStatus.Infeed1;
   IF #_w1 THEN
       #CycleSendData.Event[#Index].EventTimeStamp := #DateTime;
       #CycleSendData.Event[#Index].EventType := 27;
       #Index := #Index + 1;
   END_IF;
   #_w2 := NOT #I_SubZoneStatus.Infeed1 AND #Memory[32];   // falling edge
   #Memory[32] := #I_SubZoneStatus.Infeed1;
   IF #_w2 THEN
       #CycleSendData.Event[#Index].EventTimeStamp := #DateTime;
       #CycleSendData.Event[#Index].EventType := 28;
       #Index := #Index + 1;
   END_IF;
   IF #Index >= #MaxIndex THEN GOTO EndOfRecordReached; END_IF;
END_REGION

REGION Network 35: **** 4.4 - Machine Status - Calculated **** Register Time events - Infeed2 Start/stop
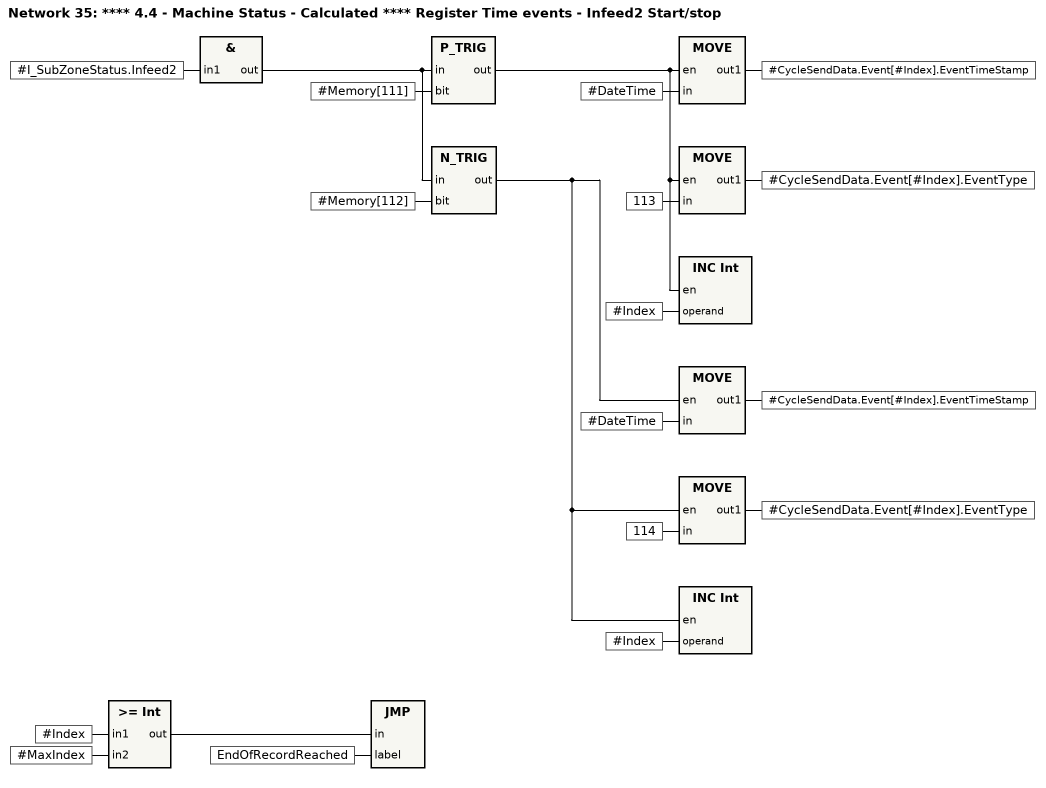
   #_w1 := #I_SubZoneStatus.Infeed2 AND NOT #Memory[111];   // rising edge
   #Memory[111] := #I_SubZoneStatus.Infeed2;
   IF #_w1 THEN
       #CycleSendData.Event[#Index].EventTimeStamp := #DateTime;
       #CycleSendData.Event[#Index].EventType := 113;
       #Index := #Index + 1;
   END_IF;
   #_w2 := NOT #I_SubZoneStatus.Infeed2 AND #Memory[112];   // falling edge
   #Memory[112] := #I_SubZoneStatus.Infeed2;
   IF #_w2 THEN
       #CycleSendData.Event[#Index].EventTimeStamp := #DateTime;
       #CycleSendData.Event[#Index].EventType := 114;
       #Index := #Index + 1;
   END_IF;
   IF #Index >= #MaxIndex THEN GOTO EndOfRecordReached; END_IF;
END_REGION

REGION Network 36: **** 4.4 - Machine Status - Calculated **** Register Time events - Infeed3 Start/stop
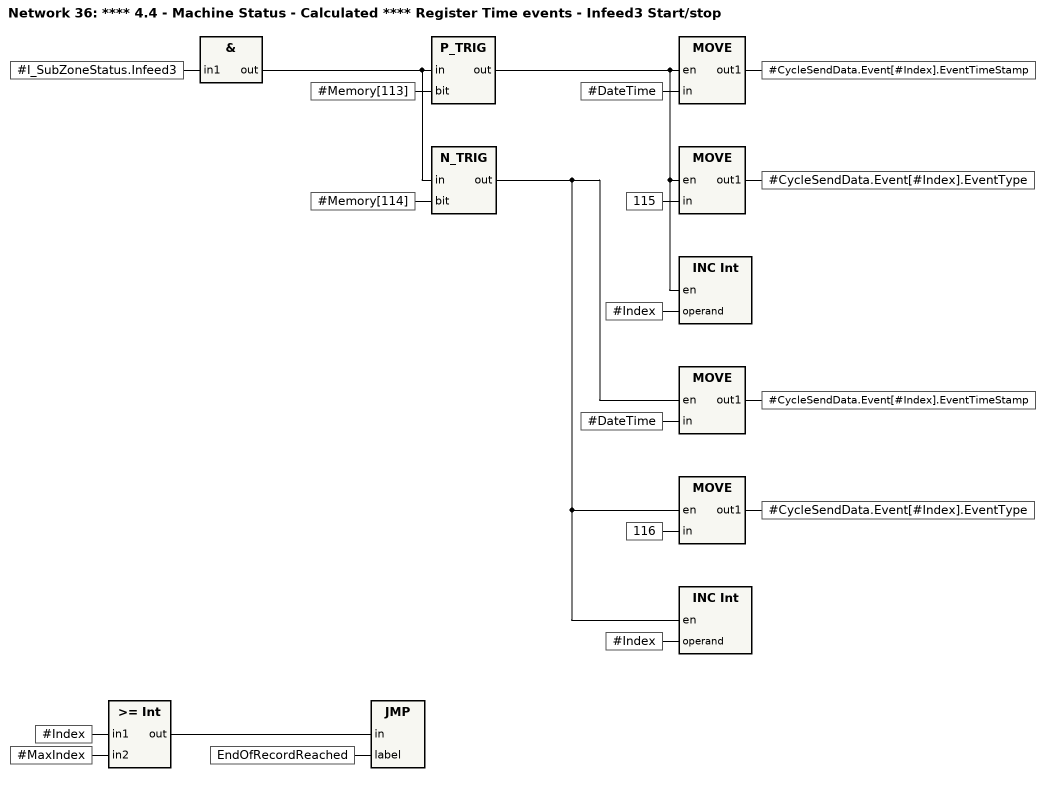
   #_w1 := #I_SubZoneStatus.Infeed3 AND NOT #Memory[113];   // rising edge
   #Memory[113] := #I_SubZoneStatus.Infeed3;
   IF #_w1 THEN
       #CycleSendData.Event[#Index].EventTimeStamp := #DateTime;
       #CycleSendData.Event[#Index].EventType := 115;
       #Index := #Index + 1;
   END_IF;
   #_w2 := NOT #I_SubZoneStatus.Infeed3 AND #Memory[114];   // falling edge
   #Memory[114] := #I_SubZoneStatus.Infeed3;
   IF #_w2 THEN
       #CycleSendData.Event[#Index].EventTimeStamp := #DateTime;
       #CycleSendData.Event[#Index].EventType := 116;
       #Index := #Index + 1;
   END_IF;
   IF #Index >= #MaxIndex THEN GOTO EndOfRecordReached; END_IF;
END_REGION

REGION Network 37: **** 4.4 - Machine Status - Calculated **** Register Time events - Infeed4 Start/stop
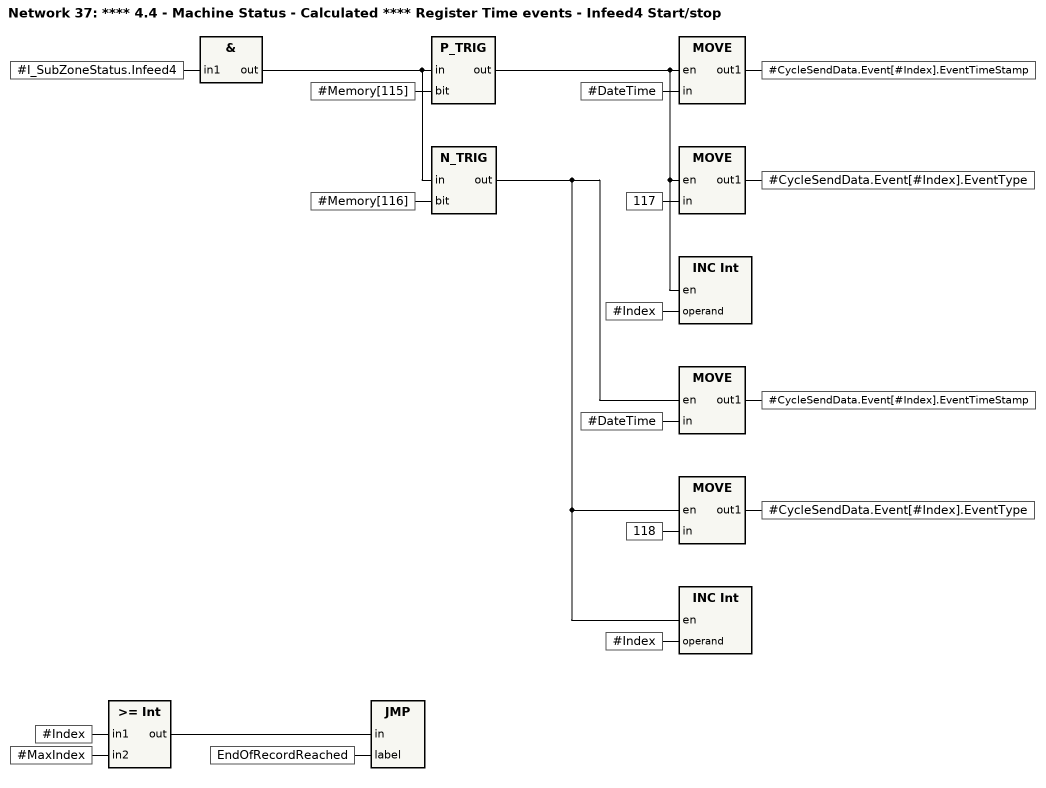
   #_w1 := #I_SubZoneStatus.Infeed4 AND NOT #Memory[115];   // rising edge
   #Memory[115] := #I_SubZoneStatus.Infeed4;
   IF #_w1 THEN
       #CycleSendData.Event[#Index].EventTimeStamp := #DateTime;
       #CycleSendData.Event[#Index].EventType := 117;
       #Index := #Index + 1;
   END_IF;
   #_w2 := NOT #I_SubZoneStatus.Infeed4 AND #Memory[116];   // falling edge
   #Memory[116] := #I_SubZoneStatus.Infeed4;
   IF #_w2 THEN
       #CycleSendData.Event[#Index].EventTimeStamp := #DateTime;
       #CycleSendData.Event[#Index].EventType := 118;
       #Index := #Index + 1;
   END_IF;
   IF #Index >= #MaxIndex THEN GOTO EndOfRecordReached; END_IF;
END_REGION

REGION Network 38: **** 4.4 - Machine Status - Calculated **** Register Time events - Infeed5 Start/stop
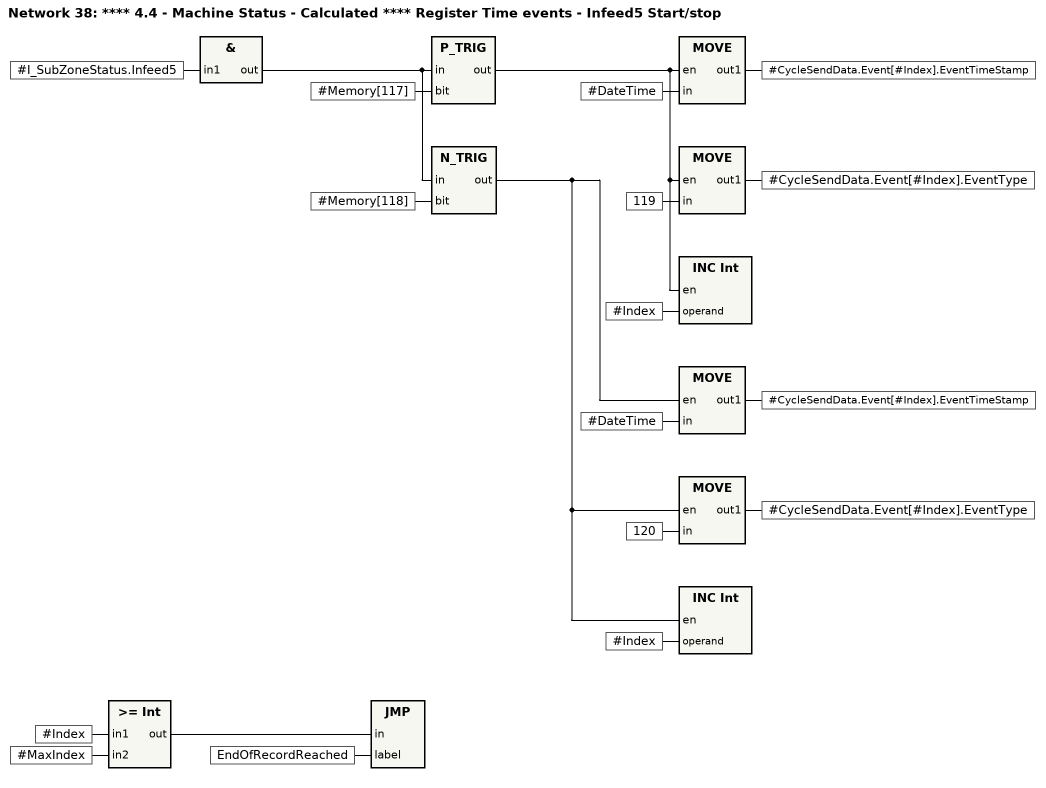
   #_w1 := #I_SubZoneStatus.Infeed5 AND NOT #Memory[117];   // rising edge
   #Memory[117] := #I_SubZoneStatus.Infeed5;
   IF #_w1 THEN
       #CycleSendData.Event[#Index].EventTimeStamp := #DateTime;
       #CycleSendData.Event[#Index].EventType := 119;
       #Index := #Index + 1;
   END_IF;
   #_w2 := NOT #I_SubZoneStatus.Infeed5 AND #Memory[118];   // falling edge
   #Memory[118] := #I_SubZoneStatus.Infeed5;
   IF #_w2 THEN
       #CycleSendData.Event[#Index].EventTimeStamp := #DateTime;
       #CycleSendData.Event[#Index].EventType := 120;
       #Index := #Index + 1;
   END_IF;
   IF #Index >= #MaxIndex THEN GOTO EndOfRecordReached; END_IF;
END_REGION

REGION Network 39: **** 4.4 - Machine Status - Calculated **** Register Time events - Waiting Process Work Start/stop
